# B&R Automation Studio project MotionTestBenchMaster (part 25)

#### Types.typ - Local data types
```iecst
TYPE
	MNM_AdjustmentStep :
		( (*V4.A.A.1.7.0*)
		MNM_AdjWaitStart := 100,
		MNM_AdjHornBlow := 110,
		MNM_AdjAxisStopping := 140,
		MNM_AdjFillerFootbarSettingPos := 200,
		MNM_AdjRinserFootbarSettingPos := 210,
		MNM_AdjDoserFootbarSettingPos := 220,
		MNM_AdjCapperSettingPos := 230,
		MNM_AdjCrownerSettingPos := 240,
		MNM_AdjCapGreasingSettingPos := 250, (*V4.A.A.1.7.0*)
		MNM_AdjAxisStart := 300,
		MNM_AdjAxisWaitStop := 310,
		MNM_AdjAxisPosStart := 400,
		MNM_AdjAxisPosWaitStop := 410,
		MNM_AdjAxisStopped := 500,
		MNM_AdjFault := 9999
		);
	MNM_AutoStep :
		(
		MNM_AutoWaitStart := 100,
		MNM_AutoHornBlow := 110,
		MNM_AutoMachineStart := 120,
		MNM_AutoMachineRunningEmpty := 131,
		MNM_AutoMachineRunningFull := 132,
		MNM_AutoMachineRunning := 133,
		MNM_AutoMachineColceaPashing := 134,
		MNM_AutoMachineStarWheel2Phasing := 137,
		MNM_AutoMachineRinserPashing := 136,
		MNM_AutoMachineStarWheel1Pashing := 135,
		MNM_AutoMachineStopping := 140,
		MNM_AutoSmr1OpHornBlow := 210,
		MNM_AutoSmr1OpMachineStart := 220,
		MNM_AutoSmr1OpMachineStopping := 240,
		MNM_AutoVortexCalibIdle := 300,
		MNM_AutoVortexCalibHornBlow := 310,
		MNM_AutoVortexCalibPosStart := 320,
		MNM_AutoVortexCalibPosWaitStop := 340,
		MNM_AutoStepFmcHornBlow := 410,
		MNM_AutoStepFmcStart := 420,
		MNM_AutoStepFmcWaitStop := 440,
		MNM_AutoStepHornBlow := 510,
		MNM_AutoStepStart := 520,
		MNM_AutoStepWaitStop := 540,
		MNM_AutoFootboardHornBlow := 610,
		MNM_AutoFootboardStart := 620,
		MNM_AutoFootboardWaitStop := 640,
		MNM_AutoCapperPosHornBlow := 710,
		MNM_AutoCapperPosStart := 720,
		MNM_AutoCapperPosWaitStop := 740,
		MNM_AutoCapperPosWaitStopAux := 741, (*V4.A.A.1.6.12h*)
		MNM_AutoCapperFinePosStart := 750,
		MNM_AutoCapperFinePosWaitStop := 760,
		MNM_AutoFillingValvePosHornBlow := 810,
		MNM_AutoFillingValvePosStart := 820,
		MNM_AutoFillingValvePosWaitStop := 830,
		MNM_AutoCheckFillerInletHorn := 1010,
		MNM_AutoCheckFillerInletStart := 1011,
		MNM_AutoCheckFillerInletStop := 1012,
		MNM_AutoCheckFillerTangencyHorn := 1020,
		MNM_AutoCheckFillerTangencyStart := 1021,
		MNM_AutoCheckFillerTangencyStop := 1022,
		MNM_AutoCheckFillerOutletHorn := 1030,
		MNM_AutoCheckFillerOutletStart := 1031,
		MNM_AutoCheckFillerOutletStop := 1032,
		MNM_AutoCheckCapsReleaseHorn := 1040,
		MNM_AutoCheckCapsReleaseStart := 1041,
		MNM_AutoCheckCapsReleaseStop := 1042,
		MNM_AutoFillerHalfPosConfig := 1043, (*v999*)
		MNM_AutoFillerHalfPosHornBlow := 1044, (*v999*)
		MNM_AutoFillerHalfAxisStart := 1045, (*v999*)
		MNM_AutoFillerHalfWaitStop := 1046, (*v999*)
		MNM_AutoFillerHalfStopped := 1047, (*v999*)
		MNM_AutoFillerReversePosConfig := 1048, (*v999*)
		MNM_AutoFillerReversePosHornBlow := 1049, (*v999*)
		MNM_AutoFillerReverseAxisStart := 1050, (*v999*)
		MNM_AutoFillerReverseWaitStop := 1051, (*v999*)
		MNM_AutoFillerReverseStopped := 1052, (*v999*)
		MNM_AutoFillSecondHalfPosConfig := 1053,
		MNM_AutoFillSecondHalfRevPosConf,
		MNM_AutoFault := 9999
		);
	MNM_AutoCombiStep :
		(
		MNM_AutoCombiInit := 0,
		MNM_AutoCombiBFWaitStart := 100,
		MNM_AutoCombiBLFWaitStart := 101,
		MNM_AutoCombiBAFWaitStart := 102, (*V4.A.A.1.7.0*)
		MNM_AutoCombiHornBlow := 110,
		MNM_AutoCombiSyncroStart := 120,
		MNM_AutoCombiMachineReadyToRun := 121,
		MNM_AutoCombiMachineRunningFull := 131,
		MNM_AutoCombiMachineRunningEmpty := 132,
		MNM_AutoCombiMachineFixEmptying := 135,
		MNM_AutoCombiMachineStopping := 140,
		MNM_AutoCombiFault := 9999
		);
	MNM_JogStep :
		(
		MNM_JogWaitStart := 400,
		MNM_JogHornBlow := 410,
		MNM_JogMachineStart := 420,
		MNM_JogMachineRunning := 430,
		MNM_JogMachineStopping := 440,
		MNM_JogFault := 9999
		);
	MNM_JogCombiStep :
		(
		MNM_JogCombiWaitStart := 400,
		MNM_JogCombiHornBlow := 410,
		MNM_JogCombiSyncroStart := 420,
		MNM_JogCombiMachineReadyToRun := 421,
		MNM_JogCombiMachineStart := 422,
		MNM_JogCombiMachineRunning := 430,
		MNM_JogCombiMachineStopping := 440,
		MNM_JogCombiFault := 9999
		);
	MNM_MultiStep :
		(
		MNM_MultiModeSelection := 0,
		MNM_MultiAutoWaitStart := 100,
		MNM_MultiAutoHornBlow := 110,
		MNM_MultiAutoMachineStart := 120,
		MNM_MultiAutoMachineRunning := 130,
		MNM_MultiAutoMachineStopping := 140,
		MNM_MultiVortexCalibIdle := 300,
		MNM_MultiVortexCalibHornBlow := 310,
		MNM_MultiVortexCalibPosStart := 320,
		MNM_MultiVortexCalibPosWaitStop := 340,
		MNM_MultiStepFmcHornBlow := 410,
		MNM_MultiStepFmcStart := 420,
		MNM_MultiStepFmcWaitStop := 440,
		MNM_MultiStepHornBlow := 510,
		MNM_MultiStepStart := 520,
		MNM_MultiStepWaitStop := 540,
		MNM_MultiFootboardHornBlow := 610,
		MNM_MultiFootboardStart := 620,
		MNM_MultiFootboardWaitStop := 640,
		MNM_MultiCapperPosHornBlow := 710,
		MNM_MultiCapperPosStart := 720,
		MNM_MultiCapperPosWaitStop := 740,
		MNM_MultiCapperFinePosStart := 750,
		MNM_MultiCapperFinePosWaitStop := 760,
		MNM_MultiJogWaitStart := 1400,
		MNM_MultiJogHornBlow := 1410,
		MNM_MultiJogMachineStart := 1420,
		MNM_MultiJogMachineRunning := 1430,
		MNM_MultiJogMachineStopping := 1440,
		MNM_MultiSlowMotionWaitStart := 1500,
		MNM_MultiSlowMotionHornBlow := 1510,
		MNM_MultiSlowMotionStart := 1520,
		MNM_MultiSlowMotionRunning := 1530,
		MNM_MultiSlowMotionStopping := 1540,
		MNM_MultiFault := 9999
		);
	MNM_InletConveyorVFD :
		( (*1.6(*Master nuovo*)
		MNM_InCvrIdle := 0,
		MNM_InCvrAuto := 100,
		MNM_InCvrAutoOption := 110,
		MNM_InCvrAutoFixSpeed := 210,
		MNM_InCvrAutoRampDown := 300,
		MNM_InCvrCleaning := 400,
		MNM_InCvrFault := 9999
		);
	MNM_OutletConveyorVFD :
		( (*1.6*)
		MNM_OutCvrIdle := 0,
		MNM_OutCvrAuto := 100,
		MNM_OutCvrAutoOption := 110,
		MNM_OutCvrAutoFixSpeed := 210,
		MNM_OutCvrAutoRampDown := 300,
		MNM_OutCvrCleaning := 400,
		MNM_OutCvrFault := 9999
		);
	VAR_FixSpeed_Type : 	STRUCT
		Module : USINT; (*0: All Module (Only coupled)
1: Inlet module
2: Filler module
3: Outlet module
9: All module (Uncupled) (Not interruptible)*)
		Interruptible : BOOL;
		Req : BOOL;
		Value : REAL;
		Reached : BOOL;
		CmpMode : USINT;
		Active : BOOL;
	END_STRUCT;
	VAR_ModuleSpeed_Type : 	STRUCT
		Machine : REAL;
		Inlet : REAL;
		Filler : REAL;
		Outlet : REAL;
	END_STRUCT;
END_TYPE
```

#### MNM_Devices.var - Local variables
```iecst
(*MOTORS*)
VAR
	_InCvrFC280 : Motor_FC280_Vfd;(*Master nuovo*)
	_OutCvrFC280 : Motor_FC280_Vfd; (*Outfeed Conveyor*)
	_InCvr : Motor_Vfd;(*Master nuovo*)
	_OutCvr : Motor_Vfd; (*Outfeed Conveyor*)
END_VAR
(*DIGITAL INSTRUMENTS*)
VAR
	_241DSE : Digital_Obj; (*Spot safety*)
	_230DSE : Digital_Obj; (*Spot safety*)
	_236DSE : Digital_Obj; (*Outlet obstructed*)
END_VAR
(*INLET CANS SENSOR*)
VAR
	InletSafetyLow1 : Digital_Obj;
	InletSafetyHigh1 : Digital_Obj;
	InletSafetyLow2 : Digital_Obj;
	InletSafetyHigh2 : Digital_Obj;
END_VAR
(*MOTORS FANS*)
(*Filler*)
VAR
	FillerFanMain : MotionFan_Obj;
	FillerFanIn1 : MotionFan_Obj;
	FillerFanIn2 : MotionFan_Obj;
	FillerFanIn3 : MotionFan_Obj;
	FillerFanIn4 : MotionFan_Obj;
	FillerFanIn5 : MotionFan_Obj;
	FillerFanIn6 : MotionFan_Obj;
	FillerFanIn7 : MotionFan_Obj;
	FillerFanIn8 : MotionFan_Obj;
	FillerFanIn9 : MotionFan_Obj;
	FillerFanIn10 : MotionFan_Obj;
	FillerFanOut1 : MotionFan_Obj;
	FillerFanOut2 : MotionFan_Obj;
	FillerFanOut3 : MotionFan_Obj;
	FillerFanOut4 : MotionFan_Obj;
	FillerFanOut5 : MotionFan_Obj;
END_VAR
(*Seamer*)
VAR
	OutletFanMain : MotionFan_Obj;
	OutletFanIn1 : MotionFan_Obj;
	OutletFanIn2 : MotionFan_Obj;
	OutletFanIn3 : MotionFan_Obj;
	OutletFanIn4 : MotionFan_Obj;
	OutletFanOut1 : MotionFan_Obj;
	OutletFanOut2 : MotionFan_Obj;
	OutletFanOut3 : MotionFan_Obj;
	OutletFanOut4 : MotionFan_Obj;
END_VAR
```

#### Package Logical/05_MNM/MNM/0520_InletConveyor - Conveyor: motori nastri Ingresso Macchina

#### InletConveyorVar_VFD.st
```iecst
ACTION InletConveyorVar_VFD:
//	VAR_MNM_ConveyorProduction	:= MC_InputOutput.Network.Filler.Status.ModuleRunning OR OPS.DataOut.FlrModeSelectorJog;
//	VAR_MNM_ConveyorClean		:= COP.DataOut.RcpActive;
END_ACTION
```

#### InletConveyorSeq_VFD.st
```iecst
ACTION InletConveyorSeq_Run_VFD:

	VAR_MNM_InCvrAlarm			:= ALR[7029].Active OR ALR[7031].Active OR ALR[7032].Active;
	_InCvrFC280.IN_AutoCnd			:= FALSE;
	_InCvrFC280.IN_AutoSpeed		:= 0.0;

	//Speed Linearization
	FB_ScalConveyorInlet(
	x	:= MC_InputOutput.Network.Machine.Status.ActualSpeed,
	x1	:= 0.0,
	y1	:= 0.0,
	x2	:= MC_InputOutput.Network.Machine.Status.MachineMaxSpeed * 1.1,
	y2	:= _InCvrFC280.IN_FrequencyMax + (_InCvrFC280.IN_FrequencyMax * HMI_PAR_1._160 / 100.0) * 1.1,
	);

	//State Management
	CASE VAR_MNM_InletConveyorSeq_VFD OF
		MNM_InCvrIdle:
			IF MNM.DataOut.MachineRunning AND NOT COP.DataOut.RcpActive AND NOT OPS.DataOut.FlrModeSelectorAdjustment THEN
				VAR_MNM_InletConveyorSeq_VFD := MNM_InCvrAuto;
			ELSIF COP.DataOut.RcpActive THEN
				_InCvrFC280.IN_AutoCnd	:= TRUE;
				VAR_MNM_InletConveyorSeq_VFD := MNM_InCvrCleaning;
			ELSIF VAR_MNM_InCvrAlarm THEN
				VAR_MNM_InletConveyorSeq_VFD := MNM_InCvrFault;
			END_IF

		MNM_InCvrAuto:

			_InCvrFC280.IN_AutoCnd		:= FB_ScalConveyorInlet.y>0.0;
			_InCvrFC280.IN_AutoSpeed	:= FB_ScalConveyorInlet.y;

			IF NOT MNM.DataOut.MachineRunning THEN
				VAR_MNM_InletConveyorSeq_VFD	:= MNM_InCvrIdle;
			ELSIF VAR_MNM_InCvrAlarm THEN
				VAR_MNM_InletConveyorSeq_VFD	:= MNM_InCvrFault;
			END_IF

		MNM_InCvrCleaning:
			_InCvrFC280.IN_AutoCnd		:= MC_InputOutput.Network.Machine.Status.MachineRunning;
			_InCvrFC280.IN_AutoSpeed	:= 10.0;

			IF NOT COP.DataOut.RcpActive THEN
				VAR_MNM_InletConveyorSeq_VFD	:= MNM_InCvrIdle;
			ELSIF VAR_MNM_InCvrAlarm THEN
				VAR_MNM_InletConveyorSeq_VFD	:= MNM_InCvrFault;
			END_IF

		MNM_InCvrFault:
			IF AID.DataOut.Reset THEN
				VAR_MNM_InletConveyorSeq_VFD := MNM_InCvrIdle;
			END_IF
	END_CASE

	TMR_TON_MNM_InCvrFix	(IN:= (VAR_MNM_InletConveyorSeq_VFD = MNM_InCvrAutoFixSpeed), PT := t#120s);
	TMR_TON_MNM_InCvrRamp	(IN:= (VAR_MNM_InletConveyorSeq_VFD = MNM_InCvrAutoRampDown), PT := t#5s);
END_ACTION
```

#### InletConveyorMotors_VFD.st
```iecst
ACTION InletConveyorMotors_VFD:
//	_InCvr(//Management with FC302
//	IN_Enable		:= OPS.DataOut.EnableDrive,
//	IN_AutoCnd		:= _InCvr.IN_AutoCnd,
//	IN_FrequencyMin	:= 0.0,
//	IN_FrequencyMax	:= 100.0,
//	IN_ManEn		:= TRUE,
//	IN_MaskEn		:= TRUE,
//	IN_Reset		:= AID.DataOut.Reset,
//	IN_HMIAutoForce	:= NOT HMI_SS2P[SS2P_HMI_DeviceEnable].ON,
//	IN_QuickStopCmd	:= NOT OPS.DataOut.EnableDrive,
//	IN_CoastingCmd	:= FALSE,
//	IN_ScaleMax		:= 100.0,
//	HMI_Danfoss		:= HMI_VFD_InCvr,
//	HMI_Motor		:= HMI_InCvr,
//	IO_Danfoss		:= IO_VFD_InCvr,
//	IO_Motor		:= IO_InCvr
//	);

	_InCvrFC280(
	IN_Enable		:= OPS.DataOut.EnableDrive,
	IN_AutoCnd		:= _InCvrFC280.IN_AutoCnd,
	IN_FrequencyMin	:= 0.0,
	IN_FrequencyMax	:= 100.0,
	IN_ManEn		:= TRUE,
	IN_MaskEn		:= TRUE,
	IN_Reset		:= AID.DataOut.Reset,
	IN_HMIAutoForce	:= NOT HMI_SS2P[SS2P_HMI_DeviceEnable].ON,
	IN_QuickStopCmd	:= NOT OPS.DataOut.EnableDrive,
	IN_CoastingCmd	:= FALSE,
	IN_ScaleMax		:= 100.0,
	HMI_Danfoss		:= HMI_VFD_InCvr,
	HMI_Motor		:= HMI_InCvr,
	IO_DanfossFC280	:= IO_VFD_InCvrFC280,
	IO_MotorFC280	:= IO_InCvrFC280
	);

END_ACTION
```

#### InletConveyorDataOut_VFD.st
```iecst
ACTION InletConveyorDataOut_VFD:
//	IF _InCvr.OUT_ActualFrequency > 0 THEN
//		MNM.DataOut.OutletSpeed := (((_InCvr.OUT_ActualFrequency / 100.0) * MC_InputOutput.Network.Machine.Status.ActualSpeed) / 60.0);
//	ELSE
//		MNM.DataOut. := 0.0 ;
//	END_IF
END_ACTION
```

#### InletConveyorAlarm_VFD.st
```iecst
ACTION InletConveyorAlarm_VFD:
//
//	ALR[7029].Active		:= _InCvr.OUT_OverloadFault;//Management with FC302
//	ALR[7031].Active		:= _InCvr.OUT_IsolatedFault;//Management with FC302
//	ALR[7032].Active		:= _InCvr.OUT_DriveFault;//Management with FC302

	ALR[7029].Active		:= _InCvrFC280.OUT_OverloadFault;
	ALR[7031].Active		:= _InCvrFC280.OUT_IsolatedFault;
	ALR[7032].Active		:= _InCvrFC280.OUT_DriveFault;
END_ACTION
```

#### InletConveyorHMI.st
```iecst
ACTION InletConveyorHMI:
	IF TNK.DataOut.ProdMode AND NOT TNK.DataOut.StartUp THEN
		HMI_ContainerFallInlet1	:= (InletSafetyLow1.OUT AND NOT InletSafetyHigh1.OUT) OR (NOT InletSafetyLow1.OUT AND InletSafetyHigh1.OUT);
		HMI_ContainerFallInlet2	:= (InletSafetyLow2.OUT AND NOT InletSafetyHigh2.OUT) OR (NOT InletSafetyLow2.OUT AND InletSafetyHigh2.OUT);
		HMI_NoContainerInlet1	:= (NOT InletSafetyLow1.OUT AND NOT InletSafetyHigh1.OUT);
		HMI_NoContainerInlet2	:= (NOT InletSafetyLow2.OUT AND NOT InletSafetyHigh2.OUT);
	ELSE
		HMI_ContainerFallInlet1	:= FALSE;
		HMI_ContainerFallInlet2	:= FALSE;
		HMI_NoContainerInlet1	:= FALSE;
		HMI_NoContainerInlet1	:= FALSE;
	END_IF
END_ACTION
```

#### InletConveyorAlarm.st
```iecst
ACTION InletConveyorAlarm:
	IF InletSafetyLow1.OUT_OffDelayed AND InletSafetyHigh1.OUT_OffDelayed AND TNK.DataOut.ProdMode AND NOT TNK.DataOut.StartUp AND CvoFlr.InfeedConveyorRunning THEN
		ALR[4618].Active	:= TRUE;   //TRUE; //COLLAUDO
	ELSE
		ALR[4618].Active	:= FALSE;
	END_IF

	IF InletSafetyLow2.OUT_OffDelayed AND InletSafetyHigh2.OUT_OffDelayed AND TNK.DataOut.ProdMode AND NOT TNK.DataOut.StartUp THEN
		ALR[4619].Active	:= TRUE;
	ELSIF AID.DataOut.Reset THEN
		ALR[4619].Active	:= FALSE;
	END_IF

	IF SFT.DataOut.ContainersBlock1 THEN
		IF TON_ContainerInletSafety1.Q AND TNK.DataOut.ProdMode AND NOT TNK.DataOut.StartUp THEN
			ALR[4620].Active	:= TRUE;
		ELSIF AID.DataOut.Reset THEN
			ALR[4620].Active	:= FALSE;
		END_IF
	ELSE
		IF ((InletSafetyLow1.OUT AND NOT InletSafetyHigh1.OUT) OR (NOT InletSafetyLow1.OUT AND InletSafetyHigh1.OUT)) AND TNK.DataOut.ProdMode AND NOT TNK.DataOut.StartUp THEN
			ALR[4620].Active	:= TRUE;
		ELSIF IO_PB_ResetInlet1.ON THEN
			ALR[4620].Active	:= FALSE;
		END_IF
	END_IF
	TON_ContainerInletSafety1.IN := ((InletSafetyLow1.OUT AND NOT InletSafetyHigh1.OUT) OR (NOT InletSafetyLow1.OUT AND InletSafetyHigh1.OUT));
	TON_ContainerInletSafety1.PT := REAL_TO_TIME((1/(MC_InputOutput.Network.Machine.Status.ActualSpeed/3600))*1000 );
	TON_ContainerInletSafety1();

	IO_PB_ResetInlet1.LampON := ALR[4620].Active AND AID.DataOut.Blink1Hz;

	IF ((InletSafetyLow2.OUT AND NOT InletSafetyHigh2.OUT) OR (NOT InletSafetyLow2.OUT AND InletSafetyHigh2.OUT)) AND TNK.DataOut.ProdMode AND NOT TNK.DataOut.StartUp THEN
		ALR[4621].Active	:= TRUE;
	ELSIF IO_PB_ResetInlet2.ON THEN
		ALR[4621].Active	:= FALSE;
	END_IF

	MNM.DataOut.LackInlet1 := ALR[4618].Active OR ALR[4620].Active;
	MNM.DataOut.LackInlet2 := ALR[4619].Active OR ALR[4621].Active;

	ALR[4600].Active	:= NOT IO_LimitTorqueBlowerTransfer.DI_Input;

END_ACTION
```

#### InletConveyor_Hardware_CFG.st
```iecst
ACTION InletConveyor_Hardware_CFG:
	(*****SENSORS*****)
	InletSafetyLow1.IN_ConfigPresent	:= TRUE;
	InletSafetyLow1.IN_OffDelay			:= t#200ms;
	InletSafetyLow1.IN_OnDelay			:= t#200ms;
	InletSafetyLow1.IN_SwitchDelay		:= t#0ms;

	InletSafetyHigh1.IN_ConfigPresent	:= TRUE;
	InletSafetyHigh1.IN_OffDelay		:= t#200ms;
	InletSafetyHigh1.IN_OnDelay			:= t#200ms;
	InletSafetyHigh1.IN_SwitchDelay		:= t#0ms;

	InletSafetyLow2.IN_ConfigPresent	:= FALSE;
	InletSafetyLow2.IN_OffDelay			:= t#200ms;
	InletSafetyLow2.IN_OnDelay			:= t#200ms;
	InletSafetyLow2.IN_SwitchDelay		:= t#0ms;

	InletSafetyHigh2.IN_ConfigPresent	:= FALSE;
	InletSafetyHigh2.IN_OffDelay		:= t#200ms;
	InletSafetyHigh2.IN_OnDelay			:= t#200ms;
	InletSafetyHigh2.IN_SwitchDelay		:= t#0ms;

//	(*****MOTORS*****)//For Inverter Model FC302, old Hardware standard
//	_InCvr.IN_ConfigPresent			:= FALSE;
//	_InCvr.IN_SafetyCtrlEn			:= TRUE;
//	_InCvr.IN_Simulation			:= FALSE;
//	_InCvr.IN_FBKDelay				:= t#1200ms;

	(*****MOTORS*****)//For Inverter Model FC280, new Hardware standard
	_InCvrFC280.IN_ConfigPresent	:= TRUE;
	_InCvrFC280.IN_SafetyCtrlEn		:= TRUE;
	_InCvrFC280.IN_Simulation		:= FALSE;
	_InCvrFC280.IN_FBKDelay			:= t#1200ms;

END_ACTION
```

#### InletConveyorDigitalIn.st
```iecst
ACTION InletConveyorDigitalIn:
	InletSafetyLow1(
	IN_ConfigPresent	:= InletSafetyLow1.IN_ConfigPresent,
	IN_Alarm			:= TRUE,
	IN_Reset			:= AID.DataOut.Reset,
	IO					:= IO_InletSafetyLow1,
	HMI					:= HMI_InletSafetyLow1
	);

	InletSafetyHigh1(
	IN_ConfigPresent	:= InletSafetyHigh1.IN_ConfigPresent,
	IN_Alarm			:= TRUE,
	IN_Reset			:= AID.DataOut.Reset,
	IO					:= IO_InletSafetyHigh1,
	HMI					:= HMI_InletSafetyHigh1
	);

	InletSafetyLow2(
	IN_ConfigPresent	:= InletSafetyLow2.IN_ConfigPresent,
	IN_Alarm			:= TRUE,
	IN_Reset			:= AID.DataOut.Reset,
	IO					:= IO_InletSafetyLow2,
	HMI					:= HMI_InletSafetyLow2
	);

	InletSafetyHigh2(
	IN_ConfigPresent	:= InletSafetyHigh2.IN_ConfigPresent,
	IN_Alarm			:= TRUE,
	IN_Reset			:= AID.DataOut.Reset,
	IO					:= IO_InletSafetyHigh2,
	HMI					:= HMI_InletSafetyHigh2
	);
END_ACTION
```

#### InletConveyorInterchange.st - not listed in the package file held
```iecst
ACTION InletConveyorInterchange:

END_ACTION
```

#### Package Logical/05_MNM/MNM/0530_OutletConveyor - Conveyor: motori nastri Uscita Macchina

#### OutletConveyor_Hardware_CFG.st
```iecst
ACTION OutletConveyor_Hardware_CFG:
	(*****MOTORS*****)//For Inverter Model FC302, old Hardware standard
//	_OutCvr.IN_ConfigPresent	:= FALSE;
//	_OutCvr.IN_SafetyCtrlEn		:= TRUE;
//	_OutCvr.IN_Simulation		:= FALSE;
//	_OutCvr.IN_FBKDelay			:= t#1200ms;

	(*****MOTORS*****)//For Inverter Model FC280, new Hardware standard
	_OutCvrFC280.IN_ConfigPresent	:= TRUE;
	_OutCvrFC280.IN_SafetyCtrlEn		:= TRUE;
	_OutCvrFC280.IN_Simulation		:= FALSE;
	_OutCvrFC280.IN_FBKDelay			:= t#1200ms;
	(*****SENSORS*****)
	// Exit Spot #1
	_230DSE.IN_ConfigPresent	:= TRUE;
	_230DSE.IN_Alarm			:= TRUE;
	_230DSE.IN_OffDelay			:= t#0s;
	_230DSE.IN_OnDelay			:= t#500ms;
	_230DSE.IN_SwitchDelay		:= t#0ms;
	// Outlet Conveyor Guide
	_236DSE.IN_ConfigPresent	:= FALSE;
	_236DSE.IN_Alarm			:= TRUE;
	_236DSE.IN_OffDelay			:= t#0s;
	_236DSE.IN_OnDelay			:= t#500ms;
	_236DSE.IN_SwitchDelay		:= t#0ms;

END_ACTION
```

#### OutletConveyorVar_VFD.st
```iecst
ACTION OutletConveyorVar_VFD:
	VAR_MNM_ConveyorProduction	:= MNM.DataOut.MachineRunning AND NOT COP.DataOut.RcpActive OR OPS.DataOut.FlrModeSelectorJog; //Montanarini: a Heuft serve il nastro in movimento quando la macchina gira	---	NOT SFT.DataOut.OutletConveyorEmpty OR NOT SFT.DataOut.MachineEmpty OR OPS.DataOut.FlrModeSelectorJog;
	VAR_MNM_ConveyorClean		:= COP.DataOut.RcpActive;
END_ACTION
```

#### OutletConveyorSeq_VFD.st
```iecst
ACTION OutletConveyorSeq_Run_VFD:
	//VAR_MNM_OutCvrAlarm			:= 	AID.DataOut.ALR.Bit.ALR_MS_NormalStop OR AID.DataOut.ALR.Bit.ALR_MS_QuickStop OR AID.DataOut.ALR.Bit.ALR_MS_NormalWithJog OR
	//								AID.DataOut.ALR.Bit.ALR_MS_QuickWithJog OR AID.DataOut.ALR.Bit.ALR_CSR_StopAfterEmptying;

	VAR_MNM_OutCvrAlarm		:= ALR[4633].Active OR ALR[4638].Active OR ALR[7039].Active OR ALR[7041].Active OR ALR[7042].Active;
	_OutCvr.IN_AutoCnd			:= FALSE;
	_OutCvr.IN_AutoSpeed		:= 0.0;

	//VAR_MNM_OptionNoGripper -> To be setted
	VAR_MNM_OptionNoGripper := TRUE;//VAR_MNM_OptionNoGripper := TRUE means that the outlet starwheel is without gripper //V4.A.A.1.6.6
									//VAR_MNM_OptionNoGripper := FALSE means that the outlet starwheel is with gripper //V4.A.A.1.6.6

	//Speed Linearization
	FB_ScalConveyor(
	x	:= MC_InputOutput.Network.Machine.Status.ActualSpeed,
	x1	:= 0.0,
	y1	:= 0.0,
	x2	:= MC_InputOutput.Network.Machine.Status.MachineMaxSpeed * 1.1,
	y2	:= _OutCvrFC280.IN_FrequencyMax + (_OutCvrFC280.IN_FrequencyMax * HMI_PAR_1._162 / 100.0) * 1.1,
	);

	//Speed Limit Threshold
	VAR_MNM_OutCvrFixSpeedLimit := MC_InputOutput.Network.Machine.Status.ActualSpeed > 10000.0;

	//Fixed Speed Calculation
	IF EDGEPOS(VAR_MNM_OutCvrFixSpeedLimit) OR EDGENEG(VAR_MNM_OutCvrFixSpeedLimit) THEN
		VAR_MNM_OutCvrFixSpeed		:= FB_ScalConveyor.y;
	END_IF

	//Fixed Speed Calculation in case of data loss
	IF VAR_MNM_OutCvrFixSpeed = 0 THEN
		VAR_MNM_OutCvrFixSpeed		:= 20.0;
	END_IF

	//State Management
	CASE VAR_MNM_OutletConveyorSeq_VFD OF
		MNM_OutCvrIdle:
			IF VAR_MNM_ConveyorProduction THEN//v1.61
				VAR_MNM_OutletConveyorSeq_VFD := MNM_OutCvrAuto;
			ELSIF VAR_MNM_ConveyorClean THEN
				_OutCvr.IN_AutoCnd	:= TRUE;
				VAR_MNM_OutletConveyorSeq_VFD := MNM_OutCvrCleaning;
			ELSIF VAR_MNM_OutCvrAlarm THEN
				VAR_MNM_OutletConveyorSeq_VFD := MNM_OutCvrFault;
			END_IF

		MNM_OutCvrAuto:

			_OutCvr.IN_AutoCnd		:= FB_ScalConveyor.y>0.0;//V4.A.A.1.6.6
			_OutCvr.IN_AutoSpeed	:= FB_ScalConveyor.y;

			IF NOT VAR_MNM_ConveyorProduction THEN
				VAR_MNM_OutletConveyorSeq_VFD	:= MNM_OutCvrIdle;
			ELSIF VAR_MNM_ConveyorProduction AND VAR_MNM_OptionNoGripper AND VAR_MNM_OutCvrFixSpeedLimit THEN//v1.61
				VAR_MNM_OutletConveyorSeq_VFD := MNM_OutCvrAutoOption;//v1.61
			ELSIF VAR_MNM_OutCvrAlarm THEN
				VAR_MNM_OutletConveyorSeq_VFD	:= MNM_OutCvrFault;
			END_IF

		MNM_OutCvrAutoOption:

			_OutCvr.IN_AutoCnd		:= FB_ScalConveyor.y>0.0;//V4.A.A.1.6.6
			_OutCvr.IN_AutoSpeed	:= FB_ScalConveyor.y;

			IF NOT VAR_MNM_ConveyorProduction OR (NOT VAR_MNM_OutCvrFixSpeedLimit AND NOT MC_InputOutput.Network.Machine.Commands.MachineStart) THEN
				VAR_MNM_OutletConveyorSeq_VFD	:= MNM_OutCvrAutoFixSpeed;
			ELSIF VAR_MNM_OutCvrAlarm THEN
				VAR_MNM_OutletConveyorSeq_VFD	:= MNM_OutCvrFault;
			END_IF

		MNM_OutCvrAutoFixSpeed:
			_OutCvr.IN_AutoCnd			:= FB_ScalConveyor.y>0.0;//V4.A.A.1.6.6
			TMR_TON_MNM_OutCvrFix.IN 	:= TRUE;

			IF MC_InputOutput.Network.Machine.Commands.MachineStart OR VAR_MNM_OutCvrFixSpeedLimit THEN
				_OutCvr.IN_AutoSpeed 		:= FB_ScalConveyor.y;
			ELSIF NOT VAR_MNM_OutCvrFixSpeedLimit AND NOT MC_InputOutput.Network.Machine.Commands.MachineStart THEN
				_OutCvr.IN_AutoSpeed 		:= VAR_MNM_OutCvrFixSpeed;
			END_IF

			IF MC_InputOutput.Network.Machine.Commands.MachineStart AND VAR_MNM_ConveyorProduction THEN
				VAR_MNM_OutletConveyorSeq_VFD	:= MNM_OutCvrAuto;
			ELSIF TMR_TON_MNM_OutCvrFix.Q THEN
				VAR_MNM_OutletConveyorSeq_VFD	:= MNM_OutCvrAutoRampDown;
				VAR_MNM_OutCvrRampDwStart		:= _OutCvr.IN_AutoSpeed;
			ELSIF VAR_MNM_OutCvrAlarm THEN
				VAR_MNM_OutletConveyorSeq_VFD	:= MNM_OutCvrFault;
			END_IF

		MNM_OutCvrAutoRampDown:
			_OutCvr.IN_AutoCnd			:= TRUE;
			_OutCvr.IN_AutoSpeed 		:= VAR_MNM_OutCvrRampDwStart -
											(VAR_MNM_OutCvrRampDwStart * (UDINT_TO_REAL(TIME_TO_UDINT(TMR_TON_MNM_OutCvrRamp.ET))) /
											(UDINT_TO_REAL(TIME_TO_UDINT(TMR_TON_MNM_OutCvrRamp.PT))));
			TMR_TON_MNM_OutCvrRamp.IN 	:= TRUE;

			IF MC_InputOutput.Network.Machine.Commands.MachineStart AND VAR_MNM_ConveyorProduction THEN
				VAR_MNM_OutletConveyorSeq_VFD	:= MNM_OutCvrAuto;
			ELSIF TMR_TON_MNM_OutCvrRamp.Q THEN
				VAR_MNM_OutletConveyorSeq_VFD	:= MNM_OutCvrIdle;
			ELSIF VAR_MNM_OutCvrAlarm THEN
				VAR_MNM_OutletConveyorSeq_VFD	:= MNM_OutCvrFault;
			END_IF

		MNM_OutCvrCleaning:
			_OutCvr.IN_AutoCnd		:= MC_InputOutput.Network.Machine.Status.MachineRunning;
			_OutCvr.IN_AutoSpeed	:= 10.0;

			IF NOT VAR_MNM_ConveyorClean THEN
				VAR_MNM_OutletConveyorSeq_VFD	:= MNM_OutCvrIdle;
			ELSIF VAR_MNM_OutCvrAlarm THEN
				VAR_MNM_OutletConveyorSeq_VFD	:= MNM_OutCvrFault;
			END_IF

		MNM_OutCvrFault:
			IF AID.DataOut.Reset THEN
				VAR_MNM_OutletConveyorSeq_VFD := MNM_OutCvrIdle;
			END_IF
	END_CASE

	TMR_TON_MNM_OutCvrFix	(IN:= (VAR_MNM_OutletConveyorSeq_VFD = MNM_OutCvrAutoFixSpeed), PT := t#120s);//<<Change this time to decide how long the conveyour runs after the last bottle or machine stop.
	TMR_TON_MNM_OutCvrRamp	(IN:= (VAR_MNM_OutletConveyorSeq_VFD = MNM_OutCvrAutoRampDown), PT := t#5s);
END_ACTION
```

#### OutletConveyorMotors_VFD.st
```iecst
ACTION OutletConveyorMotors_VFD:
//	_OutCvr(//Management with FC302
//	IN_Enable		:= OPS.DataOut.EnableDrive,
//	IN_AutoCnd		:= _OutCvr.IN_AutoCnd,
//	IN_FrequencyMin	:= 0.0,
//	IN_FrequencyMax	:= 100.0,
//	IN_ManEn		:= TRUE,
//	IN_MaskEn		:= TRUE,
//	IN_Reset		:= AID.DataOut.Reset,
//	IN_HMIAutoForce	:= NOT HMI_SS2P[SS2P_HMI_DeviceEnable].ON,
//	IN_QuickStopCmd	:= NOT OPS.DataOut.EnableDrive,
//	IN_CoastingCmd	:= FALSE,
//	IN_ScaleMax		:= 100.0,
//	HMI_Danfoss		:= HMI_VFD_OutCvr,
//	HMI_Motor		:= HMI_OutCvr,
//	IO_Danfoss		:= IO_VFD_OutCvr,
//	IO_Motor		:= IO_OutCvr
//	);

	_OutCvrFC280.IN_AutoCnd 	:= _OutCvr.IN_AutoCnd;
	_OutCvrFC280.IN_AutoSpeed	:= _OutCvr.IN_AutoSpeed;	//Montanarini: appoggio velocità

	_OutCvrFC280(
	IN_Enable		:= OPS.DataOut.EnableDrive,
	IN_AutoCnd		:= _OutCvrFC280.IN_AutoCnd,
	IN_FrequencyMin	:= 0.0,
	IN_FrequencyMax	:= 100.0,
	IN_ManEn		:= TRUE,
	IN_MaskEn		:= TRUE,
	IN_Reset		:= AID.DataOut.Reset,
	IN_HMIAutoForce	:= NOT HMI_SS2P[SS2P_HMI_DeviceEnable].ON,
	IN_QuickStopCmd	:= NOT OPS.DataOut.EnableDrive,
	IN_CoastingCmd	:= FALSE,
	IN_ScaleMax		:= 100.0,
	HMI_Danfoss		:= HMI_VFD_OutCvr,
	HMI_Motor		:= HMI_OutCvr,
	IO_DanfossFC280		:= IO_VFD_OutCvrFC280,
	IO_MotorFC280		:= IO_OutCvrFC280
	);

END_ACTION
```

#### OutletConveyorDataOut_VFD.st
```iecst
ACTION OutletConveyorDataOut_VFD:
	IF _OutCvrFC280.OUT_ActualFrequency > 0 THEN
		MNM.DataOut.OutletSpeed := (((_OutCvrFC280.OUT_ActualFrequency / 100.0) * MC_InputOutput.Network.Machine.Status.ActualSpeed) / 60.0);
	ELSE
		MNM.DataOut.OutletSpeed := 0.0 ;
	END_IF
END_ACTION
```

#### OutletConveyorAlarm_VFD.st
```iecst
ACTION OutletConveyorAlarm_VFD:
//	ALR[7039].Active		:= _OutCvr.OUT_OverloadFault;//Management with FC302
//	ALR[7041].Active		:= _OutCvr.OUT_IsolatedFault//Management with FC302
//	ALR[7042].Active		:= _OutCvr.OUT_DriveFault//Management with FC302

	ALR[7039].Active		:= _OutCvrFC280.OUT_OverloadFault;
	ALR[7041].Active		:= _OutCvrFC280.OUT_IsolatedFault;
	ALR[7042].Active		:= _OutCvrFC280.OUT_DriveFault;

	ALR[4638].Active	:= _236DSE.OUT_Alarm;
	ALR[4633].Active	:= _230DSE.OUT_Alarm;

END_ACTION
```

#### OutletConveyorMotors_Motion.st
```iecst
ACTION OutletConveyorMotors_Motion:
	MC_InputOutput.Network.Filler.Parameters.InletConveyorKs	:= HMI_PAR_1._160;
	MC_InputOutput.Network.Filler.Parameters.OutletConveyorKs	:= HMI_PAR_1._162;
	MC_InputOutput.Network.Outlet.Parameters.ConveyorKs		:= HMI_PAR_1._162;
END_ACTION
```

#### OutletConveyorAlarm_Motion.st
```iecst
ACTION OutletConveyorAlarm_Motion:
	IF NOT IO_OutCvr.DI_ManSwitchON THEN
		ALR[7041].Active	:= TRUE;
	ELSIF AID.DataOut.Reset THEN
		ALR[7041].Active	:= FALSE;
	END_IF

	ALR[4638].Active	:= _236DSE.OUT_Alarm;//v1.7.2
	ALR[4633].Active	:= _230DSE.OUT_Alarm;//v1.7.2

END_ACTION
```

#### OutletConveyorDataOut_Motion.st
```iecst
ACTION OutletConveyorDataOut_Motion:
	MNM.DataOut.OutletSpeed := ((MC_InputOutput.Network.Machine.Status.ActualSpeed / 60.0) * (1 + MC_InputOutput.Network.Outlet.Parameters.ConveyorKs / 100.0)) * LREAL_TO_REAL(CFG_MC.Mechanical.MachineStep / 1000.0) * 10.0;
END_ACTION
```

#### OutletConveyorDigitalIn.st
```iecst
ACTION OutletConveyorDigitalIn:
	_230DSE(
	IN_ConfigPresent	:= _230DSE.IN_ConfigPresent,
	IN_Reset			:= AID.DataOut.Reset,
	IN_MaskEn			:= FALSE,
	IN_WaitOn			:= TRUE,
	IN_AlarmOffReq		:= TRUE,
	IO					:= IO_230DSE,
	HMI					:= HMI_230DSE
	);

	_236DSE(
	IN_ConfigPresent	:= _236DSE.IN_ConfigPresent,
	IN_Reset			:= AID.DataOut.Reset,
	IN_MaskEn			:= FALSE,
	IN_WaitOn			:= TRUE,
	IN_AlarmOffReq		:= TRUE,
	IO					:= IO_236DSE,
	HMI					:= HMI_236DSE
	);
END_ACTION
```

#### OutletConveyorInterchange.st
```iecst
ACTION OutletConveyorInterchange:
(***************************      Alarms Standard        ****************************************)
	ALR[4626].Active	:= ((NOT CvoFlr.InfeedContainersLoadEnabled AND NOT CvoFlr.Req_Empty AND NOT SkdFlr.EndProduction) AND TNK.DataOut.ProdMode AND NOT TNK.DataOut.StartUp); //OR CvoFlr.Req_Empty;
	ALR[4629].Active	:= NOT CvoFlr.InfeedConveyorRunning AND TNK.DataOut.ProdMode AND NOT TNK.DataOut.StartUp;
	ALR[4632].Active	:= NOT CvoFlr.OutletConveyorRunning AND TNK.DataOut.ProdMode AND NOT TNK.DataOut.StartUp;
	ALR[4635].Active	:= CvoFlr.RejectTableFull AND TNK.DataOut.ProdMode AND NOT TNK.DataOut.StartUp;
	ALR[4636].Active	:= FALSE;//MasterBottle
	//ALR[4636].Active	:= CvoFlr.OutletConveyorLowSpeed AND TNK.DataOut.ProdMode AND NOT TNK.DataOut.StartUp;//PET(*Master nuovo*)
	ALR[4637].Active	:= NOT CvoFlr.OutletContainersLoadEnabled AND TNK.DataOut.ProdMode AND NOT TNK.DataOut.StartUp;
END_ACTION
```

#### OutletConveyorHMI.st
```iecst
ACTION OutletConveyorHMI:
	IF TNK.DataOut.ProdMode AND NOT TNK.DataOut.StartUp THEN
		HMI_OutletFull	:= CvoFlr.OutletConveyorLowSpeed OR NOT CvoFlr.OutletContainersLoadEnabled;
	ELSE
		HMI_OutletFull	:= FALSE;
	END_IF
END_ACTION
```

#### MNM_DataOut.st
```iecst
ACTION MNM_DataOut:
	MNM.DataOut.HornFlrRequest		:= VAR_MNM_HornFlrRequest;

	MNM.DataOut.ReadyForVortexCalib	:= VAR_MNM_AutoVortexCalibActive;

	MNM.DataOut.ReadyForCoupling	:= MC_InputOutput.Network.Machine.Status.EnableCombi;

	MNM.DataOut.FixSpeedRequest 	:= VAR_MNM_FixSpeedReq;

	MNM.DataOut.COPInletContBlockSpeedReached	:= VAR_FixSpeed[10].Reached;

	MNM.DataOut.MachineRunning		:= SEL(MC_InputOutput.Network.Machine.Status.MultiModalityActive, MC_InputOutput.Network.Machine.Status.MachineRunning, MC_InputOutput.Network.Filler.Status.ModuleRunning); //V1.0
	MNM.DataOut.RinserAxisDisabled    	:= MC_InputOutput.Network.Filler.Status.RinserAxisDisabled;//V4.A.A.1.7.0
	MNM.DataOut.DoserAxisDisabled		:= MC_InputOutput.Network.Filler.Status.DoserAxisDisabled;//v999hema
	MNM.DataOut.FillerAxisDisabled		:= MC_InputOutput.Network.Filler.Status.FillerAxisDisabled;//v999hema
	IF EDGEPOS(IO_PB_FlStart.ON)	OR EDGENEG(IO_PB_FlStop.ON)	THEN
		MNM.DataOut.OperatorPresence	:= 	TRUE;
	END_IF

END_ACTION
```

#### MNM_Alarm.st
```iecst
ACTION MNM_Alarm:

	ALR[7018].Active		:= (MC_InputOutput.Network.Machine.Status.ActualSpeed >
								(MC_InputOutput.Network.Machine.Status.MachineMaxSpeed + (MC_InputOutput.Network.Machine.Status.MachineMaxSpeed * 8.0 / 100.0))) AND MC_InputOutput.Network.Machine.Status.AutoCombiModalityActive;

	ALR[7019].Active		:= MC_InputOutput.Network.Machine.Status.ActualSpeed > (HMI_PAR_1._020 + (HMI_PAR_1._020 * 5.0 / 100.0));

	//v4 200.2.0 eliminata logica

	ALR[7155].Active	:= MC_InputOutput.Network.Machine.Exceptions.PowerSupplyLowMachineException; //V4.A.A.1.6.13
	ALR[7156].Active    := NOT IO_MNM_PowerSupply1Overload.DI_Input; //V4.A.A.1.6.13
	ALR[7157].Active	:= NOT IO_MNM_PowerSupply2Overload.DI_Input; //V4.A.A.1.6.13

	//V4.A.A.1.6.13
	ALR[7170].Active	:= (HMI_PAM_1._403 = 0) AND (HMI_201CPC.ConfigPresent OR HMI_202CPC.ConfigPresent);
	ALR[7171].Active	:= (HMI_PAM_1._407 = 0) AND CFG_Par.ClosingUnit.Capper.Present;
	ALR[7173].Active	:= (HMI_PAM_1._415 = 0) AND (HMI_PAO_2._176 <> 0);
	ALR[7174].Active 	:= (HMI_PAM_1._419 = 0) AND HMI_201CPB.ConfigPresent;
	ALR[7175].Active	:= (HMI_PAM_1._423 = 0) AND CFG_Par.ClosingUnit.Crowner.Present;
	ALR[7176].Active	:= (HMI_PAM_1._427 = 0) AND FALSE; //NOT USED AT THE MOMENT
	ALR[7177].Active	:= (HMI_PAM_1._431 = 0) AND (CFG_Par.FCI.Filltec OR CFG_Par.FCI.FTSystem OR CFG_Par.FCI.Heuft OR CFG_Par.FCI.Pressco OR CFG_Par.FCI.SIS OR CFG_Par.FCI.Stratec); //v999hema
	ALR[7178].Active	:= (HMI_PAM_1._435 = 0) AND CFG_Par.FCI.Heuft OR CFG_Par.FCI.Stratec;
	ALR[7179].Active	:= (HMI_PAM_1._439 = 0) AND CFG_Par.Doser.Present;

	ALR[7180].Active	:= NOT MC_InputOutput.Network.Filler.Status.FillerAbsolutePositionValid
							OR (NOT MC_InputOutput.Network.Filler.Status.RinserAbsolutePositionValid AND CFG_Par.Rinser.Present);
	//							OR (NOT MC_InputOutput.Network.Filler.Status.CapperAbsolutePositionValid AND CFG_Par.Lifting.Movements.Capper.UncouplingRequest) to be defined //V4.A.A.1.7.0
	//							OR (NOT MC_InputOutput.Network.Filler.Status.CrownerAbsolutePositionValid AND CFG_Par.Lifting.Movements.Crowner.UncouplingRequest);//V4.A.A.1.7.0

	//v4 200.2.0 eliminata logica
	ALR[7159].Active := MC_InputOutput.Network.Machine.Exceptions.FaultCamGeneration;//V.1.7.2
	// v4 200.2.0 eliminate logiche combi
END_ACTION

ACTION MNM_MotionAlarm:
	ALR[7002].Active	:= MC_InputOutput.Network.Machine.Exceptions.Fault;							//Motion -Motion Fault
	ALR[7004].Active	:= MC_InputOutput.Network.Machine.Exceptions.DcBusLowMachineException;		//Motion -DcBus voltage too low
	ALR[7005].Active	:= MC_InputOutput.Network.Machine.Exceptions.ExcessiveVelocityException;	//Motion -Excessive velocity requested
	ALR[7006].Active	:= MC_InputOutput.Network.Machine.Exceptions.ExcessiveAccException;			//Motion -Excessive acceleration requested
	ALR[7007].Active	:= MC_InputOutput.Network.Machine.Exceptions.NoAxisEnabledException;		//Motion -No Axis Enabled
	ALR[7008].Active	:= MC_InputOutput.Network.Machine.Exceptions.HomingException;				//Motion -Machine not in home
	ALR[7009].Active	:= MC_InputOutput.Network.Machine.Exceptions.BleederException;				//Motion -Bleeder error
	ALR[7013].Active	:= MC_InputOutput.Network.Machine.Exceptions.HmiChecksumException;			//Motion -HMI Checksum Error
	ALR[7014].Active	:= MC_InputOutput.Network.Machine.Exceptions.KochModuleNotReady;			//Motion -Koch Module Not ready

	IF (FillerFanIn1.OUT_Alarm		OR FillerFanIn2.OUT_Alarm		OR FillerFanIn3.OUT_Alarm		OR
		FillerFanIn4.OUT_Alarm		OR FillerFanIn5.OUT_Alarm		OR FillerFanIn6.OUT_Alarm		OR
		FillerFanIn7.OUT_Alarm		OR FillerFanIn8.OUT_Alarm		OR FillerFanIn9.OUT_Alarm		OR
		FillerFanIn10.OUT_Alarm		OR FillerFanMain.OUT_Alarm		OR FillerFanOut1.OUT_Alarm		OR
		FillerFanOut2.OUT_Alarm		OR FillerFanOut3.OUT_Alarm		OR FillerFanOut4.OUT_Alarm		OR
		FillerFanOut5.OUT_Alarm)	OR
		(OutletFanIn1.OUT_Alarm		OR OutletFanIn2.OUT_Alarm		OR OutletFanIn3.OUT_Alarm		OR
		OutletFanIn4.OUT_Alarm		OR OutletFanMain.OUT_Alarm		OR OutletFanOut1.OUT_Alarm		OR
		OutletFanOut2.OUT_Alarm		OR OutletFanOut3.OUT_Alarm		OR OutletFanOut4.OUT_Alarm)		OR
		MC_InputOutput.Network.Machine.Exceptions.FanSeamearFault THEN
		ALR[7015].Active := TRUE;	//Motion -Servoventilation Drive Error
	ELSE
		ALR[7015].Active := FALSE;	//Motion -Servoventilation Drive Error
	END_IF

	IF TMR_TON_TimeoutModality.Q THEN
		ALR[7016].Active	:= TRUE;
	ELSIF AID.DataOut.Reset THEN
		ALR[7016].Active	:= FALSE;
	END_IF

END_ACTION

ACTION MNM_MotionModuleAlarm:
	(*MASTER MODULE *)
	ALR[7470].Active	:= MC_InputOutput.Network.Machine.Status.ModuleNotInitialized;//1.7.2a
	(* FILLER MODULE *)
	ALR[7199].Active	:= MC_InputOutput.Network.Filler.Status.ModuleNotInitialized;			//Motion -Filler module not initialized

	IF NOT MC_InputOutput.Network.Filler.Status.ModuleNotInitialized THEN
		ALR[7200].Active	:= MC_InputOutput.Network.Filler.Exceptions.CarouselTrackException;		//Motion -Filler Carousel: Lag error
		ALR[7201].Active	:= MC_InputOutput.Network.Filler.Exceptions.CarouselHomeException;		//Motion -Filler Carousel: Not homed
		ALR[7202].Active	:= MC_InputOutput.Network.Filler.Exceptions.CarouselTorqueException;	//Motion -Filler Carousel: Torque limit exceeded
		ALR[7203].Active	:= MC_InputOutput.Network.Filler.Exceptions.CarouselDriveException;		//Motion -Filler Carousel: Drive error
		ALR[7204].Active	:= MC_InputOutput.Network.Filler.Exceptions.CarouselSafetyException;	//Motion -Filler Carousel: Safety violation
		ALR[7205].Active	:= MC_InputOutput.Network.Filler.Exceptions.CarouselNotInOpException;	//Motion -Filler Carousel: Not in operation

		ALR[7206].Active	:= MC_InputOutput.Network.Filler.Exceptions.Inlet01TrackException;		//Motion -Filler Inlet: Lag error
		ALR[7207].Active	:= MC_InputOutput.Network.Filler.Exceptions.Inlet01HomeException;		//Motion -Filler Inlet: Not homed
		ALR[7208].Active	:= MC_InputOutput.Network.Filler.Exceptions.Inlet01TorqueException;		//Motion -Filler Inlet: Torque limit exceeded
		ALR[7209].Active	:= MC_InputOutput.Network.Filler.Exceptions.Inlet01DriveException;		//Motion -Filler Inlet: Drive error
		ALR[7210].Active	:= MC_InputOutput.Network.Filler.Exceptions.Inlet01SafetyException;		//Motion -Filler Inlet: Safety violation
		ALR[7211].Active	:= MC_InputOutput.Network.Filler.Exceptions.Inlet01NotInOpException;	//Motion -Filler Inlet: Not in operation

		ALR[7212].Active	:= MC_InputOutput.Network.Filler.Exceptions.Inlet02TrackException;		//Motion -Filler Inlet: Lag error
		ALR[7213].Active	:= MC_InputOutput.Network.Filler.Exceptions.Inlet02HomeException;		//Motion -Filler Inlet: Not homed
		ALR[7214].Active	:= MC_InputOutput.Network.Filler.Exceptions.Inlet02TorqueException;		//Motion -Filler Inlet: Torque limit exceeded
		ALR[7215].Active	:= MC_InputOutput.Network.Filler.Exceptions.Inlet02DriveException;		//Motion -Filler Inlet: Drive error
		ALR[7216].Active	:= MC_InputOutput.Network.Filler.Exceptions.Inlet02SafetyException;		//Motion -Filler Inlet: Safety violation
		ALR[7217].Active	:= MC_InputOutput.Network.Filler.Exceptions.Inlet02NotInOpException;	//Motion -Filler Inlet: Not in operation

		ALR[7218].Active	:= MC_InputOutput.Network.Filler.Exceptions.Inlet03TrackException;		//Motion -Filler Inlet: Lag error
		ALR[7219].Active	:= MC_InputOutput.Network.Filler.Exceptions.Inlet03HomeException;		//Motion -Filler Inlet: Not homed
		ALR[7220].Active	:= MC_InputOutput.Network.Filler.Exceptions.Inlet03TorqueException;		//Motion -Filler Inlet: Torque limit exceeded
		ALR[7221].Active	:= MC_InputOutput.Network.Filler.Exceptions.Inlet03DriveException;		//Motion -Filler Inlet: Drive error
		ALR[7222].Active	:= MC_InputOutput.Network.Filler.Exceptions.Inlet03SafetyException;		//Motion -Filler Inlet: Safety violation
		ALR[7223].Active	:= MC_InputOutput.Network.Filler.Exceptions.Inlet03NotInOpException;	//Motion -Filler Inlet: Not in operation

		ALR[7224].Active	:= MC_InputOutput.Network.Filler.Exceptions.Inlet04TrackException;		//Motion -Filler Inlet: Lag error
		ALR[7225].Active	:= MC_InputOutput.Network.Filler.Exceptions.Inlet04HomeException;		//Motion -Filler Inlet: Not homed
		ALR[7226].Active	:= MC_InputOutput.Network.Filler.Exceptions.Inlet04TorqueException;		//Motion -Filler Inlet: Torque limit exceeded
		ALR[7227].Active	:= MC_InputOutput.Network.Filler.Exceptions.Inlet04DriveException;		//Motion -Filler Inlet: Drive error
		ALR[7228].Active	:= MC_InputOutput.Network.Filler.Exceptions.Inlet04SafetyException;		//Motion -Filler Inlet: Safety violation
		ALR[7229].Active	:= MC_InputOutput.Network.Filler.Exceptions.Inlet04NotInOpException;	//Motion -Filler Inlet: Not in operation

		ALR[7230].Active	:= MC_InputOutput.Network.Filler.Exceptions.Inlet05TrackException;		//Motion -Filler Inlet: Lag error
		ALR[7231].Active	:= MC_InputOutput.Network.Filler.Exceptions.Inlet05HomeException;		//Motion -Filler Inlet: Not homed
		ALR[7232].Active	:= MC_InputOutput.Network.Filler.Exceptions.Inlet05TorqueException;		//Motion -Filler Inlet: Torque limit exceeded
		ALR[7233].Active	:= MC_InputOutput.Network.Filler.Exceptions.Inlet05DriveException;		//Motion -Filler Inlet: Drive error
		ALR[7234].Active	:= MC_InputOutput.Network.Filler.Exceptions.Inlet05SafetyException;		//Motion -Filler Inlet: Safety violation
		ALR[7235].Active	:= MC_InputOutput.Network.Filler.Exceptions.Inlet05NotInOpException;	//Motion -Filler Inlet: Not in operation

		ALR[7236].Active	:= MC_InputOutput.Network.Filler.Exceptions.Inlet06TrackException;		//Motion -Filler Inlet: Lag error
		ALR[7237].Active	:= MC_InputOutput.Network.Filler.Exceptions.Inlet06HomeException;		//Motion -Filler Inlet: Not homed
		ALR[7238].Active	:= MC_InputOutput.Network.Filler.Exceptions.Inlet06TorqueException;		//Motion -Filler Inlet: Torque limit exceeded
		ALR[7239].Active	:= MC_InputOutput.Network.Filler.Exceptions.Inlet06DriveException;		//Motion -Filler Inlet: Drive error
		ALR[7240].Active	:= MC_InputOutput.Network.Filler.Exceptions.Inlet06SafetyException;		//Motion -Filler Inlet: Safety violation
		ALR[7241].Active	:= MC_InputOutput.Network.Filler.Exceptions.Inlet06NotInOpException;	//Motion -Filler Inlet: Not in operation

		ALR[7242].Active	:= MC_InputOutput.Network.Filler.Exceptions.Inlet07TrackException;		//Motion -Filler Inlet: Lag error
		ALR[7243].Active	:= MC_InputOutput.Network.Filler.Exceptions.Inlet07HomeException;		//Motion -Filler Inlet: Not homed
		ALR[7244].Active	:= MC_InputOutput.Network.Filler.Exceptions.Inlet07TorqueException;		//Motion -Filler Inlet: Torque limit exceeded
		ALR[7245].Active	:= MC_InputOutput.Network.Filler.Exceptions.Inlet07DriveException;		//Motion -Filler Inlet: Drive error
		ALR[7246].Active	:= MC_InputOutput.Network.Filler.Exceptions.Inlet07SafetyException;		//Motion -Filler Inlet: Safety violation
		ALR[7247].Active	:= MC_InputOutput.Network.Filler.Exceptions.Inlet07NotInOpException;	//Motion -Filler Inlet: Not in operation

		ALR[7248].Active	:= MC_InputOutput.Network.Filler.Exceptions.Inlet08TrackException;		//Motion -Filler Inlet: Lag error
		ALR[7249].Active	:= MC_InputOutput.Network.Filler.Exceptions.Inlet08HomeException;		//Motion -Filler Inlet: Not homed
		ALR[7250].Active	:= MC_InputOutput.Network.Filler.Exceptions.Inlet08TorqueException;		//Motion -Filler Inlet: Torque limit exceeded
		ALR[7251].Active	:= MC_InputOutput.Network.Filler.Exceptions.Inlet08DriveException;		//Motion -Filler Inlet: Drive error
		ALR[7252].Active	:= MC_InputOutput.Network.Filler.Exceptions.Inlet08SafetyException;		//Motion -Filler Inlet: Safety violation
		ALR[7253].Active	:= MC_InputOutput.Network.Filler.Exceptions.Inlet08NotInOpException;	//Motion -Filler Inlet: Not in operation

		ALR[7254].Active	:= MC_InputOutput.Network.Filler.Exceptions.Inlet09TrackException;		//Motion -Filler Inlet: Lag error
		ALR[7255].Active	:= MC_InputOutput.Network.Filler.Exceptions.Inlet09HomeException;		//Motion -Filler Inlet: Not homed
		ALR[7256].Active	:= MC_InputOutput.Network.Filler.Exceptions.Inlet09TorqueException;		//Motion -Filler Inlet: Torque limit exceeded
		ALR[7257].Active	:= MC_InputOutput.Network.Filler.Exceptions.Inlet09DriveException;		//Motion -Filler Inlet: Drive error
		ALR[7258].Active	:= MC_InputOutput.Network.Filler.Exceptions.Inlet09SafetyException;		//Motion -Filler Inlet: Safety violation
		ALR[7259].Active	:= MC_InputOutput.Network.Filler.Exceptions.Inlet09NotInOpException;	//Motion -Filler Inlet: Not in operation

		ALR[7260].Active	:= MC_InputOutput.Network.Filler.Exceptions.Inlet10TrackException;		//Motion -Filler Inlet: Lag error
		ALR[7261].Active	:= MC_InputOutput.Network.Filler.Exceptions.Inlet10HomeException;		//Motion -Filler Inlet: Not homed
		ALR[7262].Active	:= MC_InputOutput.Network.Filler.Exceptions.Inlet10TorqueException;		//Motion -Filler Inlet: Torque limit exceeded
		ALR[7263].Active	:= MC_InputOutput.Network.Filler.Exceptions.Inlet10DriveException;		//Motion -Filler Inlet: Drive error
		ALR[7264].Active	:= MC_InputOutput.Network.Filler.Exceptions.Inlet10SafetyException;		//Motion -Filler Inlet: Safety violation
		ALR[7265].Active	:= MC_InputOutput.Network.Filler.Exceptions.Inlet10NotInOpException;	//Motion -Filler Inlet: Not in operation

		ALR[7266].Active	:= MC_InputOutput.Network.Filler.Exceptions.Outlet01TrackException;		//Motion -Filler Outlet: Lag error
		ALR[7267].Active	:= MC_InputOutput.Network.Filler.Exceptions.Outlet01HomeException;		//Motion -Filler Outlet: Not homed
		ALR[7268].Active	:= MC_InputOutput.Network.Filler.Exceptions.Outlet01TorqueException;	//Motion -Filler Outlet: Torque limit exceeded
		ALR[7269].Active	:= MC_InputOutput.Network.Filler.Exceptions.Outlet01DriveException;		//Motion -Filler Outlet: Drive error
		ALR[7270].Active	:= MC_InputOutput.Network.Filler.Exceptions.Outlet01SafetyException;	//Motion -Filler Outlet: Safety violation
		ALR[7271].Active	:= MC_InputOutput.Network.Filler.Exceptions.Outlet01NotInOpException;	//Motion -Filler Outlet: Not in operation

		ALR[7272].Active	:= MC_InputOutput.Network.Filler.Exceptions.Outlet02TrackException;		//Motion -Filler Outlet: Lag error
		ALR[7273].Active	:= MC_InputOutput.Network.Filler.Exceptions.Outlet02HomeException;		//Motion -Filler Outlet: Not homed
		ALR[7274].Active	:= MC_InputOutput.Network.Filler.Exceptions.Outlet02TorqueException;	//Motion -Filler Outlet: Torque limit exceeded
		ALR[7275].Active	:= MC_InputOutput.Network.Filler.Exceptions.Outlet02DriveException;		//Motion -Filler Outlet: Drive error
		ALR[7276].Active	:= MC_InputOutput.Network.Filler.Exceptions.Outlet02SafetyException;	//Motion -Filler Outlet: Safety violation
		ALR[7277].Active	:= MC_InputOutput.Network.Filler.Exceptions.Outlet02NotInOpException;	//Motion -Filler Outlet: Not in operation

		ALR[7278].Active	:= MC_InputOutput.Network.Filler.Exceptions.Outlet03TrackException;		//Motion -Filler Outlet: Lag error
		ALR[7279].Active	:= MC_InputOutput.Network.Filler.Exceptions.Outlet03HomeException;		//Motion -Filler Outlet: Not homed
		ALR[7280].Active	:= MC_InputOutput.Network.Filler.Exceptions.Outlet03TorqueException;	//Motion -Filler Outlet: Torque limit exceeded
		ALR[7281].Active	:= MC_InputOutput.Network.Filler.Exceptions.Outlet03DriveException;		//Motion -Filler Outlet: Drive error
		ALR[7282].Active	:= MC_InputOutput.Network.Filler.Exceptions.Outlet03SafetyException;	//Motion -Filler Outlet: Safety violation
		ALR[7283].Active	:= MC_InputOutput.Network.Filler.Exceptions.Outlet03NotInOpException;	//Motion -Filler Outlet: Not in operation
	ELSIF EDGEPOS(MC_InputOutput.Network.Filler.Status.ModuleNotInitialized) THEN
		FOR VAR_i := 7200 TO 7283 DO
			ALR[VAR_i].Active := FALSE;
		END_FOR
	END_IF

	(* INLET MODULE *)
	ALR[7049].Active	:= MC_InputOutput.Network.Inlet.Status.ModuleNotInitialized;			//Motion -Inlet module not initialized

	IF NOT MC_InputOutput.Network.Inlet.Status.ModuleNotInitialized THEN
		ALR[7050].Active	:= MC_InputOutput.Network.Inlet.Exceptions.MainAxisTrackException;		//Motion -Inlet Carousel: Lag error
		ALR[7051].Active	:= MC_InputOutput.Network.Inlet.Exceptions.MainAxisHomeException;		//Motion -Inlet Carousel: Not homed
		ALR[7052].Active	:= MC_InputOutput.Network.Inlet.Exceptions.MainAxisTorqueException;		//Motion -Inlet Carousel: Torque limit exceeded
		ALR[7053].Active	:= MC_InputOutput.Network.Inlet.Exceptions.MainAxisDriveException;		//Motion -Inlet Carousel: Drive error
		ALR[7054].Active	:= MC_InputOutput.Network.Inlet.Exceptions.MainAxisSafetyException;		//Motion -Inlet Carousel: Safety violation
		ALR[7055].Active	:= MC_InputOutput.Network.Inlet.Exceptions.MainAxisNotInOpException;	//Motion -Inlet Carousel: Not in operation
	ELSIF EDGEPOS(MC_InputOutput.Network.Inlet.Status.ModuleNotInitialized) THEN
		FOR VAR_i := 7050 TO 7055 DO
			ALR[VAR_i].Active := FALSE;
		END_FOR
	END_IF

	(* OUTLET MODULE *)
	ALR[7349].Active	:= MC_InputOutput.Network.Outlet.Status.ModuleNotInitialized;			//Motion -Seamer module not initialized

	IF NOT MC_InputOutput.Network.Outlet.Status.ModuleNotInitialized THEN
		ALR[7350].Active	:= MC_InputOutput.Network.Outlet.Exceptions.MainAxisTrackException;		//Motion -Seamer Carousel: Lag error
		ALR[7351].Active	:= MC_InputOutput.Network.Outlet.Exceptions.MainAxisHomeException;		//Motion -Seamer Carousel: Not homed
		ALR[7352].Active	:= MC_InputOutput.Network.Outlet.Exceptions.MainAxisTorqueException;	//Motion -Seamer Carousel: Torque limit exceeded
		ALR[7353].Active	:= MC_InputOutput.Network.Outlet.Exceptions.MainAxisDriveException;		//Motion -Seamer Carousel: Drive error
		ALR[7354].Active	:= MC_InputOutput.Network.Outlet.Exceptions.MainAxisSafetyException;	//Motion -Seamer Carousel: Safety violation
		ALR[7355].Active	:= MC_InputOutput.Network.Outlet.Exceptions.MainAxisNotInOpException;	//Motion -Seamer Carousel: Not in operation

		ALR[7416].Active	:= MC_InputOutput.Network.Outlet.Exceptions.Outlet01TrackException;		//Motion -Seamer Carousel: Lag error
		ALR[7417].Active	:= MC_InputOutput.Network.Outlet.Exceptions.Outlet01HomeException;		//Motion -Seamer Carousel: Not homed
		ALR[7418].Active	:= MC_InputOutput.Network.Outlet.Exceptions.Outlet01TorqueException;	//Motion -Seamer Carousel: Torque limit exceeded
		ALR[7419].Active	:= MC_InputOutput.Network.Outlet.Exceptions.Outlet01DriveException;		//Motion -Seamer Carousel: Drive error
		ALR[7420].Active	:= MC_InputOutput.Network.Outlet.Exceptions.Outlet01SafetyException;	//Motion -Seamer Carousel: Safety violation
		ALR[7421].Active	:= MC_InputOutput.Network.Outlet.Exceptions.Outlet01NotInOpException;	//Motion -Seamer Carousel: Not in operation
	ELSIF EDGEPOS(MC_InputOutput.Network.Outlet.Status.ModuleNotInitialized) THEN
		FOR VAR_i := 7350 TO 7421 DO
			ALR[VAR_i].Active := FALSE;
		END_FOR
	END_IF
END_ACTION
```

#### MNM_DisableMotorManagement.st
```iecst
ACTION MNM_DisableMotorManagement:
 // in wait riabilito tutto ipotesi uno
	VAR_MNM_DefaultAxisConfig := DOS.DataOut.AllAxisEnableRequest OR (TNK.DataOut.DummyContainersDis AND TNK.DataOut.CipMode);

	IF DOS.DataOut.AxisEnableRequest AND VAR_MNM_AxisDisableStep <> 1 AND NOT DOS.DataOut.RunOnlyHemaAxisRequest THEN
		VAR_MNM_AxisDisableStep := 1;
	ELSIF DOS.DataOut.AxisDisableRequest AND VAR_MNM_AxisDisableStep <> 2 THEN
		VAR_MNM_AxisDisableStep := 2;
	ELSIF DOS.DataOut.RunOnlyHemaAxisRequest AND VAR_MNM_AxisDisableStep <> 3 THEN
		VAR_MNM_AxisDisableStep := 3;
	ELSIF DOS.DataOut.RunRinserHemaAxisRequest AND VAR_MNM_AxisDisableStep <> 4 THEN
		VAR_MNM_AxisDisableStep := 4;
	ELSIF RNS.DataOut.RunOnlyRinserAxisRequest AND VAR_MNM_AxisDisableStep <> 5 THEN
		VAR_MNM_AxisDisableStep := 5;
	ELSIF VAR_MNM_DefaultAxisConfig AND VAR_MNM_AxisDisableStep <> 0 THEN
		VAR_MNM_AxisDisableStep := 0;
	END_IF

	IF VAR_MNM_AxisConfigLoadedNumber <> VAR_MNM_AxisDisableStep OR ALR[3015].Active OR ALR[3016].Active  THEN
		VAR_MNM_NormalStop := TRUE;
	ELSIF VAR_MNM_AxisConfigLoadedNumber = VAR_MNM_AxisDisableStep THEN
		VAR_MNM_NormalStop := FALSE;
	END_IF

	CASE VAR_MNM_AxisDisableStep OF

		0: // Configuration of Motor must be disabled //Default Motor Configuration all axis are Enabled
			IF NOT MNM.DataOut.MachineRunning THEN
				memcpy( ADR(MC_InputOutput.Network.Filler.Commands.MotorDisableIndex),ADR(CFG_MC.MotorDisableConfig[0]), SIZEOF(CFG_MC.MotorDisableConfig[0]));
			END_IF
			MNM.DataOut.ConfigReqLoaded := (memcmp( ADR( MC_InputOutput.Network.Filler.Status.AxisDisabledFeedBack), ADR(CFG_MC.MotorDisableConfig[0]) ,SIZEOF(CFG_MC.MotorDisableConfig[0])) = 0);

			IF 	MNM.DataOut.ConfigReqLoaded THEN
				MNM.DataOut.ConfigReqLoaded	:= FALSE;
				VAR_MNM_AxisConfigLoadedNumber	:= 0;
			END_IF

		1:// configuration 1 request to MC , wait answer from MC program //DOSER ENABLE
			IF NOT MNM.DataOut.MachineRunning THEN
				memcpy( ADR(MC_InputOutput.Network.Filler.Commands.MotorDisableIndex),ADR(CFG_MC.MotorDisableConfig[1]), SIZEOF(CFG_MC.MotorDisableConfig[1]));
			END_IF
			MNM.DataOut.ConfigReqLoaded := (memcmp( ADR( MC_InputOutput.Network.Filler.Status.AxisDisabledFeedBack), ADR(CFG_MC.MotorDisableConfig[1]) ,SIZEOF(CFG_MC.MotorDisableConfig[1])) = 0);

			IF 	MNM.DataOut.ConfigReqLoaded AND NOT DOS.DataOut.AxisEnableRequest THEN
				MNM.DataOut.ConfigReqLoaded	:= FALSE;
				VAR_MNM_AxisConfigLoadedNumber	:= 1;
			END_IF
		2:// configuration 1 request to MC , wait answer from MC program DOSER DISABLE
			IF NOT MNM.DataOut.MachineRunning THEN
				memcpy( ADR(MC_InputOutput.Network.Filler.Commands.MotorDisableIndex),ADR(CFG_MC.MotorDisableConfig[2]), SIZEOF(CFG_MC.MotorDisableConfig[2]));
			 END_IF
			MNM.DataOut.ConfigReqLoaded := (memcmp( ADR( MC_InputOutput.Network.Filler.Status.AxisDisabledFeedBack), ADR(CFG_MC.MotorDisableConfig[2]) ,SIZEOF(CFG_MC.MotorDisableConfig[2])) = 0);

			IF 	MNM.DataOut.ConfigReqLoaded AND NOT DOS.DataOut.AxisDisableRequest THEN
				MNM.DataOut.ConfigReqLoaded	:= FALSE;
				VAR_MNM_AxisConfigLoadedNumber	:= 2;
			END_IF

		3:// configuration 1 request to MC , wait answer from MC program DOSER ONLY
			IF NOT MNM.DataOut.MachineRunning THEN
				memcpy( ADR(MC_InputOutput.Network.Filler.Commands.MotorDisableIndex),ADR(CFG_MC.MotorDisableConfig[3]), SIZEOF(CFG_MC.MotorDisableConfig[3]));
			END_IF
			MNM.DataOut.ConfigReqLoaded := (memcmp( ADR( MC_InputOutput.Network.Filler.Status.AxisDisabledFeedBack), ADR(CFG_MC.MotorDisableConfig[3]) ,SIZEOF(CFG_MC.MotorDisableConfig[3])) = 0);

			IF MNM.DataOut.ConfigReqLoaded THEN
				VAR_MNM_AxisConfigLoadedNumber	:= 3;
			END_IF

			IF 	MNM.DataOut.ConfigReqLoaded AND NOT DOS.DataOut.RunOnlyHemaAxisRequest THEN
				MNM.DataOut.ConfigReqLoaded	:= FALSE;
				VAR_MNM_AxisConfigLoadedNumber	:= 3;
			END_IF

		4:// configuration 1 request to MC , wait answer from MC program DOSER + RINSER ONLY
			IF NOT MNM.DataOut.MachineRunning THEN
				memcpy( ADR(MC_InputOutput.Network.Filler.Commands.MotorDisableIndex),ADR(CFG_MC.MotorDisableConfig[4]), SIZEOF(CFG_MC.MotorDisableConfig[4]));
			END_IF
			MNM.DataOut.ConfigReqLoaded := (memcmp( ADR( MC_InputOutput.Network.Filler.Status.AxisDisabledFeedBack), ADR(CFG_MC.MotorDisableConfig[4]) ,SIZEOF(CFG_MC.MotorDisableConfig[4])) = 0);

			IF MNM.DataOut.ConfigReqLoaded THEN
				VAR_MNM_AxisConfigLoadedNumber	:= 4;
			END_IF

			IF 	MNM.DataOut.ConfigReqLoaded AND NOT DOS.DataOut.RunRinserHemaAxisRequest THEN
				MNM.DataOut.ConfigReqLoaded	:= FALSE;
				VAR_MNM_AxisConfigLoadedNumber	:= 4;
			END_IF
		5:// configuration 1 request to MC , wait answer from MC program RINSER ONLY
			IF NOT MNM.DataOut.MachineRunning THEN
				memcpy( ADR(MC_InputOutput.Network.Filler.Commands.MotorDisableIndex),ADR(CFG_MC.MotorDisableConfig[5]), SIZEOF(CFG_MC.MotorDisableConfig[5]));
			END_IF
			MNM.DataOut.ConfigReqLoaded := (memcmp( ADR( MC_InputOutput.Network.Filler.Status.AxisDisabledFeedBack), ADR(CFG_MC.MotorDisableConfig[5]) ,SIZEOF(CFG_MC.MotorDisableConfig[5])) = 0);

			IF 	MNM.DataOut.ConfigReqLoaded AND NOT RNS.DataOut.RunOnlyRinserAxisRequest THEN
				MNM.DataOut.ConfigReqLoaded	:= FALSE;
				VAR_MNM_AxisConfigLoadedNumber	:= 5;
			END_IF
	END_CASE
END_ACTION
```

#### MNM_MachineSpeedManagemant.st
```iecst
ACTION MNM_MachineSpeedManagemant:
	VAR_ModuleSpeed.Machine	:= 0.0;
	VAR_ModuleSpeed.Inlet	:= 0.0;
	VAR_ModuleSpeed.Filler	:= 0.0;
	VAR_ModuleSpeed.Outlet	:= 0.0;

	VAR_FixSpeedActive		:= 0;
	VAR_InFixSpeedActive	:= 0;
	VAR_FlrFixSpeedActive	:= 0;
	VAR_OutFixSpeedActive	:= 0;

	IF NOT MC_InputOutput.Network.Machine.Status.MultiModalityActive THEN
		FOR iSpeed := 1 TO CST_FixSpeedMax DO
			IF VAR_FixSpeed[iSpeed].Req AND VAR_FixSpeedActive = 0 THEN
				VAR_ModuleSpeed.Machine		:= VAR_FixSpeed[iSpeed].Value;
				VAR_FixSpeedActive			:= iSpeed;
			END_IF

			IF VAR_FixSpeedActive <> 0 AND VAR_FixSpeed[iSpeed].Req THEN
				IF VAR_FixSpeed[VAR_FixSpeedActive].Interruptible THEN
					VAR_ModuleSpeed.Machine		:= VAR_FixSpeed[iSpeed].Value;
					VAR_FixSpeedActive			:= iSpeed;
				END_IF
			END_IF

			TON_ReachedDelay[iSpeed](
			IN := FC_SpeedCheck(IN_SpeedReq := VAR_FixSpeed[iSpeed].Value, IN_SpeedAct := MC_InputOutput.Network.Machine.Status.ActualSpeed, IN_Mode := VAR_FixSpeed[iSpeed].CmpMode),
			PT := t#2s
			);
			VAR_FixSpeed[iSpeed].Reached := TON_ReachedDelay[iSpeed].Q AND VAR_FixSpeed[iSpeed].Req;
		END_FOR
	ELSE
		FOR iSpeed := 1 TO CST_FixSpeedMax DO
			IF VAR_FixSpeed[iSpeed].Req AND VAR_FixSpeedActive = 0 THEN//1.7.2
				IF VAR_FixSpeed[iSpeed].Module = 1 THEN
					VAR_ModuleSpeed.Inlet	:= VAR_FixSpeed[iSpeed].Value;
					VAR_InFixSpeedActive	:= iSpeed;
				ELSIF VAR_FixSpeed[iSpeed].Module = 2 THEN
					VAR_ModuleSpeed.Filler	:= VAR_FixSpeed[iSpeed].Value;
					VAR_FlrFixSpeedActive	:= iSpeed;
				ELSIF VAR_FixSpeed[iSpeed].Module = 3 THEN
					VAR_ModuleSpeed.Outlet	:= VAR_FixSpeed[iSpeed].Value;
					VAR_OutFixSpeedActive	:= iSpeed;
				ELSIF VAR_FixSpeed[iSpeed].Module = 9 THEN
					VAR_ModuleSpeed.Inlet	:= VAR_FixSpeed[iSpeed].Value;
					VAR_ModuleSpeed.Filler	:= VAR_FixSpeed[iSpeed].Value;
					VAR_ModuleSpeed.Outlet	:= VAR_FixSpeed[iSpeed].Value;
					VAR_InFixSpeedActive	:= iSpeed;
					VAR_FlrFixSpeedActive	:= iSpeed;
					VAR_OutFixSpeedActive	:= iSpeed;
				END_IF
			END_IF

			IF VAR_InFixSpeedActive <> 0 AND VAR_FixSpeed[iSpeed].Req AND VAR_FixSpeed[iSpeed].Module = 1 THEN
				IF VAR_FixSpeed[VAR_InFixSpeedActive].Interruptible THEN
					VAR_ModuleSpeed.Inlet	:= VAR_FixSpeed[iSpeed].Value;
					VAR_InFixSpeedActive	:= iSpeed;
				END_IF
			END_IF

			IF VAR_FlrFixSpeedActive <> 0 AND VAR_FixSpeed[iSpeed].Req AND VAR_FixSpeed[iSpeed].Module = 2 THEN
				IF VAR_FixSpeed[VAR_FlrFixSpeedActive].Interruptible THEN
					VAR_ModuleSpeed.Filler	:= VAR_FixSpeed[iSpeed].Value;
					VAR_FlrFixSpeedActive	:= iSpeed;
				END_IF
			END_IF

			IF VAR_OutFixSpeedActive <> 0 AND VAR_FixSpeed[iSpeed].Req AND VAR_FixSpeed[iSpeed].Module = 3 THEN
				IF VAR_FixSpeed[VAR_OutFixSpeedActive].Interruptible THEN
					VAR_ModuleSpeed.Outlet	:= VAR_FixSpeed[iSpeed].Value;
					VAR_OutFixSpeedActive	:= iSpeed;
				END_IF
			END_IF

			IF VAR_FixSpeed[iSpeed].Module = 1 THEN
				TON_ReachedDelay[iSpeed](
				IN := FC_SpeedCheck(IN_SpeedReq := VAR_FixSpeed[iSpeed].Value, IN_SpeedAct := MC_InputOutput.Network.Inlet.Status.Velocity, IN_Mode := VAR_FixSpeed[iSpeed].CmpMode),
				PT := t#2s
				);
			END_IF

			IF VAR_FixSpeed[iSpeed].Module = 2 THEN
				TON_ReachedDelay[iSpeed](
				IN := FC_SpeedCheck(IN_SpeedReq := VAR_FixSpeed[iSpeed].Value, IN_SpeedAct := MC_InputOutput.Network.Filler.Status.Velocity, IN_Mode := VAR_FixSpeed[iSpeed].CmpMode),
				PT := t#2s
				);
			END_IF

			IF VAR_FixSpeed[iSpeed].Module = 3 THEN
				TON_ReachedDelay[iSpeed](
				IN := FC_SpeedCheck(IN_SpeedReq := VAR_FixSpeed[iSpeed].Value, IN_SpeedAct := MC_InputOutput.Network.Outlet.Status.Velocity, IN_Mode := VAR_FixSpeed[iSpeed].CmpMode),
				PT := t#2s
				);
			END_IF

			IF VAR_FixSpeed[iSpeed].Module = 9 THEN
				IF MC_InputOutput.Network.Inlet.Status.ModuleReal THEN
					TON_ReachedDelay[iSpeed].IN	:= FC_SpeedCheck(	IN_SpeedReq := VAR_FixSpeed[iSpeed].Value,
					IN_SpeedAct := MC_InputOutput.Network.Inlet.Status.Velocity,
					IN_Mode := VAR_FixSpeed[iSpeed].CmpMode);
				ELSE
					TON_ReachedDelay[iSpeed].IN := TRUE;
				END_IF

				IF MC_InputOutput.Network.Filler.Status.ModuleReal THEN
					TON_ReachedDelay[iSpeed].IN	:= FC_SpeedCheck(	IN_SpeedReq := VAR_FixSpeed[iSpeed].Value,
					IN_SpeedAct := MC_InputOutput.Network.Filler.Status.Velocity,
					IN_Mode := VAR_FixSpeed[iSpeed].CmpMode) AND TON_ReachedDelay[iSpeed].IN;
				ELSE
					TON_ReachedDelay[iSpeed].IN := TON_ReachedDelay[iSpeed].IN;
				END_IF

				IF MC_InputOutput.Network.Outlet.Status.ModuleReal THEN
					TON_ReachedDelay[iSpeed].IN	:= FC_SpeedCheck(	IN_SpeedReq := VAR_FixSpeed[iSpeed].Value,
					IN_SpeedAct := MC_InputOutput.Network.Outlet.Status.Velocity,
					IN_Mode := VAR_FixSpeed[iSpeed].CmpMode) AND TON_ReachedDelay[iSpeed].IN;
				ELSE
					TON_ReachedDelay[iSpeed].IN := TON_ReachedDelay[iSpeed].IN;
				END_IF

				TON_ReachedDelay[iSpeed](
				PT := t#2s
				);
			END_IF
			VAR_FixSpeed[iSpeed].Reached := TON_ReachedDelay[iSpeed].Q AND VAR_FixSpeed[iSpeed].Req;
		END_FOR
	END_IF

	IF VAR_FixSpeedActive = 0 THEN
		VAR_ModuleSpeed.Machine	:= DINT_TO_REAL(HMI_MNM_FlrSpeedWidget.AutoSpeedReq);
	END_IF

	IF VAR_InFixSpeedActive = 0 THEN
		VAR_ModuleSpeed.Inlet;
	END_IF

	IF VAR_FlrFixSpeedActive = 0 THEN
		VAR_ModuleSpeed.Filler	:= DINT_TO_REAL(HMI_MNM_FlrSpeedWidget.AutoSpeedReq);
	END_IF

	IF VAR_OutFixSpeedActive = 0 THEN
		VAR_ModuleSpeed.Outlet	:= DINT_TO_REAL(HMI_MNM_SmrSpeedWidget.AutoSpeedReq);
	END_IF

	IF VAR_FixSpeedActive <> 0 OR VAR_InFixSpeedActive <> 0 OR VAR_FlrFixSpeedActive <> 0 OR VAR_OutFixSpeedActive <> 0 THEN
		VAR_MNM_FixSpeedReq := TRUE;
	ELSE
		VAR_MNM_FixSpeedReq := FALSE;
	END_IF

END_ACTION
```

### Package Logical/08_RNS - Rinser: gestione Sciacquatrice

### Program Logical/08_RNS/RNS (IEC) - RNS Main Program - C#4 - 100ms

#### RNS.sfc - Cyclic code
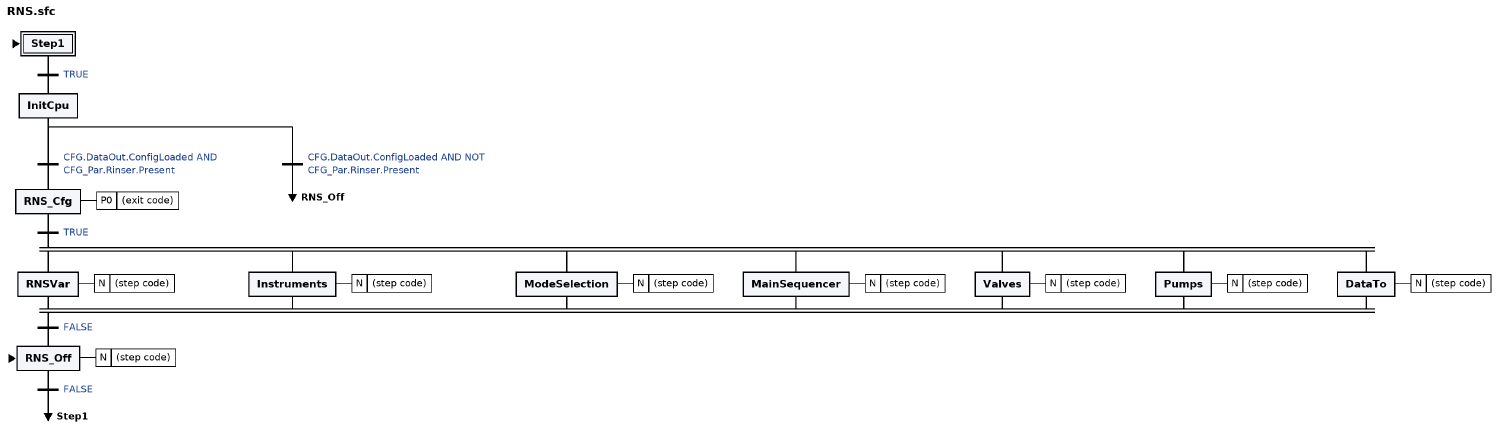
```iecst
PROGRAM _CYCLIC
INITIAL_STEP Step1:
END_STEP
TRANSITION FROM Step1 TO InitCpu:=
TRUE
END_TRANSITION
STEP InitCpu:
END_STEP
TRANSITION PRESENT FROM InitCpu TO RNS_Cfg:=
CFG.DataOut.ConfigLoaded AND CFG_Par.Rinser.Present
END_TRANSITION
TRANSITION NOT PRESENT FROM InitCpu TO RNS_Off:=
CFG.DataOut.ConfigLoaded AND NOT CFG_Par.Rinser.Present
END_TRANSITION
(* @SFCISJUMP := 'RNS_Off' *)
STEP RNS_Cfg:
END_STEP
EXIT_ACTION
RNS_Hardware_CFG;

HMI_CFG_PAC_1._201	:= TRUE;
HMI_CFG_PAC_1._202	:= TRUE;

HMI_CFG_PAM_1._014 	:= CFG_Par.Rinser.PressureNozzleControlInsertion;
HMI_CFG_PAM_1._015 	:= CFG_Par.Rinser.PressureNozzleControlContinous;
HMI_CFG_PAM_1._081 	:= CFG_Par.Rinser.PressureNozzleControlInsertion;
HMI_CFG_PAM_1._083 	:= CFG_Par.Rinser.PressureNozzleControlContinous;
HMI_CFG_PAM_1._085 	:= CFG_Par.Rinser.PressureNozzleControlContinous;
HMI_CFG_PAM_1._087 	:= CFG_Par.Rinser.PressureNozzleControlInsertion;
HMI_CFG_PAM_1._089 	:= CFG_Par.Rinser.PressureNozzleControlContinous;
HMI_CFG_PAM_1._090 	:= CFG_Par.Rinser.PressureNozzleControlInsertion;
HMI_CFG_PAM_1._091 	:= CFG_Par.Rinser.PressureNozzleControlContinous;
//RVB202 SP
HMI_CFG_PAM_1._092 	:= PTB[220].IN_ConfigPresent;
//Recovery pump speed
HMI_CFG_PAM_1._116 := PPB[209].IN_ConfigPresent;
HMI_CFG_PAM_1._117 := PPB[209].IN_ConfigPresent;
HMI_CFG_PAM_1._118 := PPB[209].IN_ConfigPresent;

HMI_CFG_PAR_1._167	:= TRUE;
HMI_CFG_PAR_1._168	:= TRUE;
HMI_CFG_PAR_1._169	:= TRUE;
HMI_CFG_PAR_1._170	:= TRUE;
HMI_CFG_PAR_1._171	:= CFG_Par.Rinser.PressureNozzleControlInsertion OR CFG_Par.Rinser.PressureNozzleControlContinous;

//HMI Buttons//V4.A.A.1.7.0
HMI_RNS_SS2P[SS2P_SelAutoMan].Visibility		:= TRUE;
HMI_RNS_SS2P[SS2P_SelProduction].Visibility		:= TRUE;
HMI_RNS_SS2P[SS2P_SelDrain].Visibility			:= TRUE;
HMI_RNS_SS2P[SS2P_SelCIP].Visibility			:= FALSE; //CFG_Par.Rinser.CipPresent;
HMI_RNS_SS2P[SS2P_RNS_InsControl].Visibility	:= CFG_Par.Rinser.PressureNozzleControlInsertion;
HMI_RNS_SS2P[SS2P_RNS_ContControl].Visibility	:= CFG_Par.Rinser.PressureNozzleControlContinous;
HMI_RNS_PB[PB_CmdStart].Visibility				:= TRUE;
HMI_RNS_PB[PB_CmdStop].Visibility				:= TRUE;

(*RNS Nozzles Data Scroll //V4.A.A.1.7.0*)
VAR_RNS_MinPageData := 0;
VAR_RNS_MaxPageData := (HMI_PAC_1._200 / 15) -1;

HMI_RNS_PB[PB_RNS_PageDown].Visibility 	:= TRUE;
HMI_RNS_PB[PB_RNS_PageUp].Visibility 	:= TRUE;

VAR_RNS_NozzleInLastPage := (HMI_PAC_1._200 MOD 15);

IF VAR_RNS_NozzleInLastPage > 0 THEN
	VAR_RNS_MaxPageData := VAR_RNS_MaxPageData + 1;
END_IF
END_ACTION
TRANSITION FROM RNS_Cfg TO (RNSVar,Instruments,ModeSelection,MainSequencer,Valves,Pumps,DataTo):=
TRUE
END_TRANSITION
STEP RNSVar:
VAR_RNS_Blink1HzEp 		:= EDGEPOS(AID.DataOut.Blink1Hz);
VAR_RNS_PBResetEp		:= EDGEPOS(AID.DataOut.Reset);
END_STEP
STEP Instruments:
RNS_InstrFlow;
RNS_InstrPress;
RNS_InstrSaf;
RNS_InstrLevel; //v1.4
END_STEP
STEP ModeSelection:
RNS_ModeSelection;
END_STEP
STEP MainSequencer:
RNS_StepManager;
RNS_StepMove;
RNS_StepConfig;
RNS_StepStatus;
END_STEP
STEP Valves:
RNS_ValvesLogic;
RNS_ValvesFB;
RNS_ModulatingValvesPID;
END_STEP
STEP Pumps:
RNS_PumpsLogic;
RNS_PumpsPID;
RNS_PumpsFB;
END_STEP
STEP DataTo:
RNS_Alarm;
RNS_HMI;
RNS_DataOut;//V4.A.A.1.7.0
END_STEP
TRANSITION FROM (RNSVar,Instruments,ModeSelection,MainSequencer,Valves,Pumps,DataTo) TO RNS_Off:=
FALSE
END_TRANSITION
STEP RNS_Off:
ST_tmp_suspend(0);
END_STEP
TRANSITION FROM RNS_Off TO Step1:=
FALSE
END_TRANSITION
(* @SFCISJUMP := 'Step1' *)
END_PROGRAM
```

#### Devices.var
```iecst
(*VALVES*)
VAR
	AVB : ARRAY[MIN_CFG_AVx..MAX_CFG_AVx] OF Valve_Dig;
END_VAR
(*INSTRUMENTS - DIGITAL*)
VAR
	FSB : ARRAY[MIN_CFG_FSx..MAX_CFG_FSx] OF Digital_Obj;
	LSB : ARRAY[MIN_CFG_LSx..MAX_CFG_LSx] OF Digital_Obj;
END_VAR
(*RINSER RELEASED CLAMPS SAFETY*)
VAR
	_202DSB : Digital_Obj;
END_VAR
(*INSTRUMENTS - ANALOGIC*)
VAR
	PTB : ARRAY[MIN_CFG_PTx..MAX_CFG_PTx] OF Analog_In;
	LTB : ARRAY[MIN_CFG_LTx..MAX_CFG_LTx] OF Analog_In; (*vRMA*)
	FTB : ARRAY[MIN_CFG_FTx..MAX_CFG_FTx] OF Analog_In;
END_VAR
(*MOTORS*)
VAR
	PPB : ARRAY[MIN_CFG_VFD_PPx..MAX_CFG_VFD_PPx] OF Motor_FC280_Vfd;
	FB_PID_PPB209 : PID_Cont;
END_VAR
```

#### Types.typ - Local data types
```iecst
TYPE
	SEQ_Type : 	STRUCT
		Step : ARRAY[0..MAX_STEP_CFG]OF SEQ_Step_Type;
		ModeActual : UINT;
		StepActual : UINT;
		TON_Time_END : BOOL;
		T_Time_END : BOOL;
		TO_Time_END : BOOL;
		Laps_Done : BOOL;
		Cycles_Done : BOOL; (*All Cycles Done*)
	END_STRUCT;
	SEQ_Step_Type : 	STRUCT  (*V4.A.A.1.7.0*)
		Jump : ARRAY[0..MAX_JUMP_CFG]OF SEQ_Jump_Type;
		Config : SEQ_StepConfig_Type;
	END_STRUCT;
	SEQ_Jump_Type : 	STRUCT  (*V4.A.A.1.7.0*)
		Condition : BOOL;
		Number : UINT;
	END_STRUCT;
	VAR_RNS_SeqActualStep_Type :
		( (*V4.A.A.1.7.0*)
		RNS_SeqWait := 0,
		RNS_SeqPrdPriming := 5,
		RNS_SeqPrdPrimingTimeOut := 6,
		RNS_SeqSystemWaitCon := 7,
		RNS_SeqSystemOnTreatment := 11,
		RNS_SeqSystemTreatmentAlr := 26,
		RNS_SeqDrain := 22,
		RNS_SeqDrainDone := 23,
		RNS_SeqCip := 24, (*v1.4*)
		RNS_SeqCop := 25, (*v1.4*)
		RNS_SeqCipStopped := 30, (*v1.4*)
		RNS_SeqControl := 70, (*V4.A.A.1.7.0*)
		RNS_SeqBypass := 90, (*V4.A.A.1.7.0*)
		RNS_SeqStopped := 40
		);
END_TYPE

(*DEVICES*)

TYPE
	SEQ_Module_Type : 	STRUCT
		Device : SEQ_Device_Type;
		Mem : SEQ_Mem_Type;
		ITC : SEQ_ITC_Type;
	END_STRUCT;
	SEQ_Mem_Type : 	STRUCT
		ContainersStop : BOOL; (*Containers Stop Control (1 = Stop)*)
		ByPassRequest : BOOL; (*Rincer ByPass Request*)
		ByPassed : BOOL; (*Rincer ByPassed*)
		WaterTreatmentControl : BOOL; (*Water Spray Continous Mode*)
		AirTreatmentControl : BOOL; (*Air Spray Control Mode*)
		ControlInsercion : BOOL; (*Spray Control Insercion Mode*)
		ControlContinous : BOOL; (*Spray Control Continous Mode*)
		InsercionDevice : BOOL; (*Spray Control Device insercion Request*)
		SpeedReductionControl : BOOL; (*Spray Control Device insercion Request*)
		CopAfterCipRequest : BOOL; (*Cop Request After CIP*)
		PBAbortEnable : BOOL; (*PB Abort Sequence Enable*)
		PBStopEnable : BOOL; (*PB Stop Sequence Enable*)
		PBStartEnable : BOOL; (*PB Start Sequence Enable*)
		NoBoNoSprayInsercion : BOOL; (*No Bottle No Spray Insercion Device for Priming Nozle Rma tes*)
	END_STRUCT;
	SEQ_Device_Type : 	STRUCT
		AVB224 : Valve_Cmd_Type;
		AVB228 : Valve_Cmd_Type; (*V4.A.A.1.7.0*)
		AVB234 : Valve_Cmd_Type; (*vrma*)
		AVB261 : Valve_Cmd_Type;
		AVB264 : Valve_Cmd_Type; (*V4.A.A.1.7.0*)
		AVB265 : Valve_Cmd_Type; (*V4.A.A.1.7.0*)
		AVB266 : Valve_Cmd_Type; (*V4.A.A.1.7.0*)
		AVB267 : Valve_Cmd_Type; (*v1.4*)
		AVB268 : Valve_Cmd_Type; (*v1.4*)
		AVB273 : Valve_Cmd_Type; (*V4.A.A.1.7.0*)
		AVB294 : Valve_Cmd_Type;
		PPB209 : Seq_Motor_Type; (*v1.4*)
		RVB202_PID : PID_Type; (*V4.A.A.1.7.0*)
		PPB209_PID : PID_Type; (*v1.4*)
		LSB209 : Digital_In_Type; (*v1.4*)
		LSB210 : Digital_In_Type; (*v1.4*)
		LSB299 : Digital_In_Type; (*v1.4*)
		LTB202 : Analog_In_Type; (*vrma*)
		FSB201 : Digital_In_Type;
		FSB220 : Digital_In_Type;
		FTB201 : Analog_In_Type; (*v1.4*)
		FTB202 : Analog_In_Type; (*V4.A.A.1.7.0*)
		PTB220 : Analog_In_Type; (*V4.A.A.1.7.0*)
		PTB270 : Analog_In_Type; (*V4.A.A.1.7.0*)
		PTB290 : Analog_In_Type;
	END_STRUCT;
	SEQ_ITC_Type : 	STRUCT
		WTT_ProductRequest : BOOL; (*Production Mode Active*)
		WTT_ProductionRunning : BOOL; (*Filler Inlet Open - Start/Stop Overpressure Pump*)
	END_STRUCT;
	Analog_In_Type : 	STRUCT
		ALR_HighLimitEn : BOOL;
		ALR_HighLimitSP : REAL;
		ALR_LowLimitEn : BOOL;
		ALR_LowLimitSP : REAL;
		SP : REAL;
		CMP : USINT;
		MinDev : REAL;
		MaxDev : REAL;
	END_STRUCT;
	Digital_In_Type : 	STRUCT
		ALR : BOOL;
		WAIT_ON : BOOL;
		WAIT_OFF : BOOL;
	END_STRUCT;
	PID_Type : 	STRUCT
		PID_Enable : BOOL; (*PID Enable Condition*)
		PID_Mode : BOOL; (*PID Mode (1 = Auto - 0 = Manual)*)
		Auto_SP_Value : REAL;
		Auto_SP_MinDev : REAL;
		Auto_SP_MaxDev : REAL;
		FIX_Value : REAL;
	END_STRUCT;
	Seq_Motor_Type : 	STRUCT
		IN_Auto : BOOL; (*PID Enable Condition*)
		IN_AutoSP : REAL;
		IN_FixOut : BOOL;
		IN_FixOutValue : REAL;
	END_STRUCT;
	Valve_Cmd_Type : 	STRUCT
		AutoCnd : BOOL;
		EnableCnd : BOOL;
	END_STRUCT;
	Motor_Cmd_Type : 	STRUCT
		AutoCnd : BOOL;
	END_STRUCT;
END_TYPE
```

#### Variables.var - Local variables
```iecst
VAR
	TOF_StatusMachineRunning : TOF;
END_VAR
(*SELECTIONS*)
VAR
	VAR_RNS_FMDProduction : BOOL;
	VAR_RNS_FMDDrain : BOOL;
	VAR_RNS_FMDCip : BOOL;
	VAR_RNS_FMDCop : BOOL;
	VAR_RNS_FMDControl : BOOL; (*v4.A.A.A.1.6.15*)
	VAR_RNS_FMDByPass : BOOL; (*v4.A.A.A.1.6.15*)
	VAR_RNS_MemPBStart : BOOL;
	VAR_RNS_MemPBStop : BOOL;
	VAR_RNS_MemPBAbort : BOOL;
	VAR_RNS_MemPBSkipForward : BOOL;
	VAR_RNS_MemSSPause : BOOL;
END_VAR
(*AUXILIARY VARIABLES*)
VAR
	VAR_RNS_Blink1HzEp : BOOL;
	VAR_RNS_PBResetEp : BOOL;
	VAR_RNS_PBSelectionEnable : BOOL;
	VAR_RNS_TankLevelMedium : BOOL; (*v1.4*)
	VAR_RNS_TankLevelTooLow : BOOL;
	VAR_RNS_TankLevelLow : BOOL;
	VAR_RNS_TankLevelHigh : BOOL;
	VAR_RNS_InletOpen : BOOL;
	VAR_RNS_InletProductIncoming : BOOL;
	VAR_RNS_InletOpenCip : BOOL; (*v4.A.A.A.1.6.15*)
	VAR_RNS_OutletOpen : BOOL;
	VAR_RNS_ProductInletSafety : BOOL;
	VAR_RNS_ProductInletSafetyDelay : BOOL;
	VAR_RNS_ForIndex : UINT;
	VAR_RNS_MinPageData : INT; (*v4.A.A.A.1.6.15*)
	VAR_RNS_MaxPageData : INT; (*v4.A.A.A.1.6.15*)
	VAR_RNS_ActPageData : INT; (*v4.A.A.A.1.6.15*)
	VAR_RNS_NozzleInLastPage : INT; (*v4.A.A.A.1.6.15*)
	VAR_RNS_IndexVis : INT; (*v4.A.A.A.1.6.15*)
	VAR_RNS_IndexAlarm : INT; (*v4.A.A.A.1.6.15*)
	VAR_RNS_ContinousAirAlarm : UINT; (*v4.A.A.A.1.6.15*)
	VAR_RNS_ContinousWaterAlarm : UINT; (*v4.A.A.A.1.6.15*)
	VAR_RNS_InsercionAirAlarm : UINT; (*v4.A.A.A.1.6.15*)
	VAR_RNS_InsercionWaterAlarm : UINT; (*v4.A.A.A.1.6.15*)
	VAR_RNS_IndexReset : INT; (*v4.A.A.A.1.6.15*)
	VAR_RNS_TotalContainerEntered : UDINT; (*v4.A.A.A.1.6.15*)
	VAR_RNS_ControlRemainder_Cont : UDINT; (*v4.A.A.A.1.6.15*)
	VAR_RNS_ControlRemainder : UDINT; (*v4.A.A.A.1.6.15*)
	VAR_RNS_AirTreatment : BOOL; (*v4.A.A.A.1.6.15*)
	VAR_RNS_WaterTreatment : BOOL; (*v4.A.A.A.1.6.15*)
	VAR_RNS_CleaningActive : BOOL; (*v4.A.A.A.1.6.15*)
	VAR_RNS_ControlModeRequest : BOOL; (*v4.A.A.A.1.6.15*)
	VAR_RNS_ControlInsercionRequest : BOOL; (*v4.A.A.A.1.6.15*)
	VAR_RNS_ControlContinousRequest : BOOL; (*v4.A.A.A.1.6.15*)
	VAR_RNS_BypassRequest : BOOL; (*v4.A.A.A.1.6.15*)
	VAR_RNS_BypassCommand : BOOL; (*v4.A.A.A.1.6.15*)
	VAR_RNS_MemDisableAxisReq : BOOL; (*//RnsDisable*)
END_VAR
(*ALARM VARIABLES*)
VAR
	VAR_RNS_AirFlowTooHigh : BOOL; (*v4.A.A.A.1.6.15*)
	VAR_RNS_AirFlowTooLow : BOOL; (*v4.A.A.A.1.6.15*)
	VAR_RNS_AirFlowLowWarning : BOOL; (*v4.A.A.A.1.6.15*)
	VAR_RNS_WaterFlowTooHigh : BOOL;
	VAR_RNS_WaterFlowTooLow : BOOL;
	VAR_RNS_WaterFlowLowWarning : BOOL; (*v4.A.A.A.1.6.15*)
	VAR_RNS_WaterFlowMissing : BOOL; (*v4.A.A.A.1.6.15*)
	VAR_RNS_BottlesNotRinse : BOOL;
	VAR_RNS_AVB_ValveFault : BOOL;
END_VAR
(*AUXILIARY TIMERS*)
VAR
	TMR_TON_TankLowLevelLost : TON;
	TMR_TON_InletSafetyDelay : TON;
	TMR_TON_AirFlowLowLimitDelay : TON; (*v4.A.A.A.1.6.15*)
	TMR_TON_WtrFlowLowLimitDelay : TON; (*v4.A.A.A.1.6.15*)
	TMR_TON_WtrFlowSwitchDelay : TON; (*v4.A.A.A.1.6.15*)
	TMR_TON_FlipWait : TON;
	TMR_TOF_FlipWork : TOF;
END_VAR
(*PID*)
VAR CONSTANT
	PID_MODE_CIP : USINT := 0;
	PID_MODE_PRD : USINT := 1;
END_VAR
VAR
	FB_PID_RVB202 : ARRAY[0..3] OF PID_Cont; (*v4.A.A.A.1.6.15*)
	FB_PID_PPB220 : ARRAY[0..3] OF PID_Cont;
END_VAR
(*SAFETY STATUS*)
VAR
	VAR_RNS_ValveEnable : BOOL;
	VAR_RNS_ValveEnableCip : BOOL; (*v4.A.A.A.1.6.15*)
	VAR_RNS_PumpEnable : BOOL;
	VAR_RNS_MotorEnable : BOOL;
	VAR_SetReset : SR; (*v1.4*)
	VAR_RNS_RVB202Auto : BOOL; (*v4.A.A.A.1.6.15*)
END_VAR
```

#### VariablesSeq.var - Local variables
```iecst
(*SEQUENCER*)
VAR
	FB_RNS_SEQ : Sequencer_v2;
	VAR_RNS_SEQ_Step : SEQ_Type;
	VAR_RNS_SEQ : SEQ_Module_Type;
	VAR_RNS_SeqProdStopAlarm : BOOL;
	VAR_RNS_SeqProdStopRequest : BOOL;
	VAR_RNS_SeqProdAbortRequest : BOOL;
	VAR_RNS_SeqCipStopAlarm : BOOL;
	VAR_RNS_SeqCipStopRequest : BOOL;
	VAR_RNS_SeqCipAbortRequest : BOOL;
	VAR_RNS_SeqDrainStopAlarm : BOOL;
	VAR_RNS_SeqDrainStopRequest : BOOL;
	VAR_RNS_SeqDrainAbortRequest : BOOL;
	VAR_RNS_SeqControlStopAlarm : BOOL; (*v4.A.A.A.1.6.15*)
	VAR_RNS_SeqControlStopRequest : BOOL; (*v4.A.A.A.1.6.15*)
	VAR_RNS_SeqControlAbortRequest : BOOL; (*v4.A.A.A.1.6.15*)
	VAR_RNS_SeqBypassStopAlarm : BOOL; (*v4.A.A.A.1.6.15*)
	VAR_RNS_SeqBypassAbortRequest : BOOL; (*v4.A.A.A.1.6.15*)
	VAR_index : UINT;
	VAR_RNS_SeqActualStep : UINT;(*v4.A.A.A.1.6.15*)
	VAR_RNS_SeqCyclesCounter : UDINT;
END_VAR
(*MODE VARIABLES*)
VAR
	VAR_RNS_ModeWait : BOOL;
	VAR_RNS_ModeProduction : BOOL;
	VAR_RNS_ModeCip : BOOL;
	VAR_RNS_ModeRinse : BOOL;
	VAR_RNS_ModeDrain : BOOL;
	VAR_RNS_ModeCop : BOOL;
	VAR_RNS_ModeControl : BOOL;(*v4.A.A.A.1.6.15*)
	VAR_RNS_ModeBypass : BOOL; (*v4.A.A.A.1.6.15*)
	VAR_RNS_MemProdDrain : BOOL;
	VAR_RNS_MemProdControl : BOOL;
	VAR_RNS_MemRinserByPassed : BOOL;(*v4.A.A.A.1.6.15*)
	VAR_RNS_MemRinserInserted : BOOL; (*v4.A.A.A.1.6.15*)
	VAR_RNS_ModeFiltersSterilization : BOOL;
	VAR_RNS_ModeDeEnergization : BOOL;
	VAR_RNS_ModeWaitOperator : BOOL;
END_VAR
(*STEP VARIABLES*)
(*Production*)
VAR
	VAR_RNS_StepProdStartUp : BOOL;
	VAR_RNS_StepProdStartUpLampCtrl : BOOL;
	VAR_RNS_StepProdStartUpLampFault : BOOL;
	VAR_RNS_StepProdProducing : BOOL;
	VAR_RNS_StepProdSprayRequest : BOOL;
	VAR_RNS_StepProdLampOnDischarge : BOOL;
	VAR_RNS_StepProdStopped : BOOL;
	VAR_RNS_StepProdAborted : BOOL;
END_VAR
(*Cip*)
VAR
	VAR_RNS_StepCipFilling : BOOL;
	VAR_RNS_StepCipCleaning : BOOL;
	VAR_RNS_StepCipDraining : BOOL;
	VAR_RNS_StepCipRecovery : BOOL;
	VAR_RNS_StepCipPipeFlooding : BOOL;
	VAR_RNS_StepCipPipeDischarge : BOOL;
	VAR_RNS_StepCipFlooding : BOOL;
	VAR_RNS_StepCipFlooded : BOOL;
	VAR_RNS_StepCipStopped : BOOL;
	VAR_RNS_StepCipAborted : BOOL;
	VAR_RNS_StepCipEnded : BOOL;
END_VAR
(*Drain*)
VAR
	VAR_RNS_StepDrainStopped : BOOL;
	VAR_RNS_StepDrainAborted : BOOL;
END_VAR
(*Control*)
VAR
	VAR_RNS_StepControl : BOOL;(*v4.A.A.A.1.6.15*)
	VAR_RNS_StepControlDone : BOOL;(*v4.A.A.A.1.6.15*)
	VAR_RNS_StepCtrlCipDone : BOOL; (*v4.A.A.A.1.6.15*)
	VAR_RNS_StepControlStopped : BOOL;(*v4.A.A.A.1.6.15*)
	VAR_RNS_StepControlAborted : BOOL;(*v4.A.A.A.1.6.15*)
END_VAR
(*By Pass*)
VAR
	VAR_RNS_StepByPassed : BOOL;(*v4.A.A.A.1.6.15*)
	VAR_RNS_StepBypassAborted : BOOL;(*v4.A.A.A.1.6.15*)
END_VAR
(*Motion*)
VAR
	VAR_RNS_StepMotorization : BOOL; (*//RnsDisable*)
END_VAR
```

#### RNS_InstrFlow.st
```iecst
ACTION RNS_InstrFlow:
//FSB201 RINSER
	FSB[201](
	IN_ConfigPresent 	:= FSB[201].IN_ConfigPresent,
	IN_Alarm 			:= TNK.DataOut.ProdMode AND MNM.DataOut.MachineRunning AND AVB[228].IN_AutoCnd,
	IN_AlarmOnReq		:= FALSE,
	IN_AlarmOffReq 		:= (AVB[228].IN_ConfigPresent AND TNK.DataOut.ProdMode AND MNM.DataOut.MachineRunning AND AVB[228].IN_AutoCnd),
	IN_SwitchDelay 		:= T#50ms,
	IN_WaitOn 			:= AVB[228].IN_AutoCnd,
	IN_WaitOff 			:= FALSE,
	IN_Reset	 		:= VAR_RNS_PBResetEp,
	IN_MaskEn 			:= TRUE,
	IO 					:= IO_FSB[201],
	HMI 				:= HMI_FSB[201]
	);

//FSB220 RINSER SPRAY FLOWSWITCH

	//Alarm Delay//V4.A.A.1.7.0
	TMR_TON_WtrFlowSwitchDelay.IN := VAR_RNS_SEQ.Device.FSB220.ALR  AND SFT.DataOut.NoBottleNoSprayActive AND VAR_RNS_InletProductIncoming;//vrma
	TMR_TON_WtrFlowSwitchDelay.PT := T#5s;
	TMR_TON_WtrFlowSwitchDelay();

	FSB[220](//V4.A.A.1.7.0
	IN_ConfigPresent 	:= FSB[220].IN_ConfigPresent,
	IN_Alarm 			:= TMR_TON_WtrFlowSwitchDelay.Q,
	IN_AlarmOnReq		:= FALSE,
	IN_AlarmOffReq 		:= TMR_TON_WtrFlowSwitchDelay.Q,
	IN_SwitchDelay 		:= T#50ms,
	IN_WaitOn 			:= VAR_RNS_SEQ.Device.FSB220.WAIT_ON,
	IN_WaitOff 			:= FALSE,
	IN_Reset	 		:= VAR_RNS_PBResetEp,
	IN_MaskEn 			:= TRUE,
	IO 					:= IO_FSB[220],
	HMI 				:= HMI_FSB[220]
	);

	IF FSB[220].OUT_Alarm THEN//V4.A.A.1.7.0
		VAR_RNS_WaterFlowMissing :=  TRUE ;
	ELSIF VAR_RNS_PBResetEp THEN
		VAR_RNS_WaterFlowMissing :=  FALSE;
	END_IF

//FTB201 RINSER FLOW TRASMITTER AIR

	//Alarm Delay
	TMR_TON_AirFlowLowLimitDelay.IN := VAR_RNS_SEQ.Device.FTB201.ALR_LowLimitEn;
	TMR_TON_AirFlowLowLimitDelay.PT := T#5s;
	TMR_TON_AirFlowLowLimitDelay();

	IF TMR_TON_AirFlowLowLimitDelay.Q THEN
		FTB[201].IN_LowLimitDelay := T#1s;
	ELSE
		FTB[201].IN_LowLimitDelay := T#5s;
	END_IF

	FTB[201](
	IN_ConfigPresent 	:= FTB[201].IN_ConfigPresent,
	IN_EngScale 		:= FTB[201].IN_EngScale,
	IN_CompareMode 		:= VAR_RNS_SEQ.Device.FTB201.CMP,
	IN_AlarmEn 			:= TRUE,
	IN_MaskEn 			:= TRUE,
	IN_Reset 			:= VAR_RNS_PBResetEp,
	IN_ActualSP 		:= VAR_RNS_SEQ.Device.FTB201.SP,
	IN_MinDev 			:= VAR_RNS_SEQ.Device.FTB201.MinDev,
	IN_MaxDev 			:= VAR_RNS_SEQ.Device.FTB201.MaxDev,
	IN_WaitDelay 		:= T#500ms,
	IN_HighLimitEn 		:= VAR_RNS_SEQ.Device.FTB201.ALR_HighLimitEn,
	IN_HighLimitSP 		:= VAR_RNS_SEQ.Device.FTB201.ALR_HighLimitSP,
	IN_HighLimitHyst 	:= 0.0,
	IN_HighLimitDelay 	:= T#1s,
	IN_LowLimitEn 		:= VAR_RNS_SEQ.Device.FTB201.ALR_LowLimitEn,
	IN_LowLimitSP 		:= VAR_RNS_SEQ.Device.FTB201.ALR_LowLimitSP,
	IN_LowLimitHyst 	:= 0.0,
	IN_LowLimitDelay 	:= FTB[201].IN_LowLimitDelay,
	IN_TotPulseWeight 	:= 0.0,
	IN_TotType 			:= 0,
	IN_PLCCounterEn 	:= FALSE,
	IN_PLCCounterSP 	:= 0.0,
	IN_PLCCounterReset	:= FALSE,
	IN_HMITotEn 		:= FALSE,
	IN_HMITotReset 		:= FALSE,
	IO 					:= IO_FTB[201],
	HMI 				:= HMI_FTB[201]
	);

	VAR_RNS_AirFlowTooHigh := FTB[201].OUT_HighLimit;

	IF FTB[201].OUT_LowLimit THEN
		VAR_RNS_AirFlowTooLow	:= TRUE;
	ELSIF VAR_RNS_PBResetEp THEN
		VAR_RNS_AirFlowTooLow	:= FALSE;
	END_IF

	VAR_RNS_AirFlowLowWarning := NOT FTB[201].OUT_SpReached AND (FTB[201].OUT_ActValue < FTB[201].IN_ActualSP);

//FTB202 RINSER FLOW TRASMITTER H2O

	//Alarm Delay
	TMR_TON_WtrFlowLowLimitDelay.IN := VAR_RNS_SEQ.Device.FTB202.ALR_LowLimitEn AND SFT.DataOut.NoBottleNoSprayActive AND VAR_RNS_InletProductIncoming;//vrma
	TMR_TON_WtrFlowLowLimitDelay.PT := T#5s;
	TMR_TON_WtrFlowLowLimitDelay();

	IF TMR_TON_WtrFlowLowLimitDelay.Q THEN
		FTB[202].IN_LowLimitDelay := T#1s;
	ELSE
		FTB[202].IN_LowLimitDelay := T#5s;
	END_IF

	FTB[202](
	IN_ConfigPresent 	:= FTB[202].IN_ConfigPresent,
	IN_EngScale 		:= FTB[202].IN_EngScale,
	IN_CompareMode 		:= VAR_RNS_SEQ.Device.FTB202.CMP,
	IN_AlarmEn 			:= TRUE,
	IN_MaskEn 			:= TRUE,
	IN_Reset 			:= VAR_RNS_PBResetEp,
	IN_ActualSP 		:= VAR_RNS_SEQ.Device.FTB202.SP,
	IN_MinDev 			:= VAR_RNS_SEQ.Device.FTB202.MinDev,
	IN_MaxDev 			:= VAR_RNS_SEQ.Device.FTB202.MaxDev,
	IN_WaitDelay 		:= T#500ms,
	IN_HighLimitEn 		:= VAR_RNS_SEQ.Device.FTB202.ALR_HighLimitEn AND SFT.DataOut.NoBottleNoSprayActive,
	IN_HighLimitSP 		:= VAR_RNS_SEQ.Device.FTB202.ALR_HighLimitSP,
	IN_HighLimitHyst 	:= 0.0,
	IN_HighLimitDelay 	:= T#1s,
	IN_LowLimitEn 		:= VAR_RNS_SEQ.Device.FTB202.ALR_LowLimitEn AND SFT.DataOut.NoBottleNoSprayActive AND VAR_RNS_InletProductIncoming,
	IN_LowLimitSP 		:= VAR_RNS_SEQ.Device.FTB202.ALR_LowLimitSP,
	IN_LowLimitHyst 	:= 0.0,
	IN_LowLimitDelay 	:= FTB[202].IN_LowLimitDelay,
	IN_TotPulseWeight 	:= 0.0,
	IN_TotType 			:= 0,
	IN_PLCCounterEn 	:= FALSE,
	IN_PLCCounterSP 	:= 0.0,
	IN_PLCCounterReset	:= FALSE,
	IN_HMITotEn 		:= FALSE,
	IN_HMITotReset 		:= FALSE,
	IO 					:= IO_FTB[202],
	HMI 				:= HMI_FTB[202]
	);

	VAR_RNS_WaterFlowTooHigh := FTB[202].OUT_HighLimit;

	IF FTB[202].OUT_LowLimit THEN
		VAR_RNS_WaterFlowTooLow	:= NOT SFT.DataOut.MachineEmpty;
	ELSIF VAR_RNS_PBResetEp THEN
		VAR_RNS_WaterFlowTooLow	:= FALSE;
	END_IF

	IF VAR_RNS_SEQ.Device.FTB202.ALR_LowLimitEn AND SFT.DataOut.NoBottleNoSprayActive AND VAR_RNS_InletProductIncoming  THEN//vrma
		VAR_RNS_WaterFlowLowWarning := NOT FTB[202].OUT_SpReached AND (FTB[202].OUT_ActValue < FTB[202].IN_ActualSP);
	ELSE
		VAR_RNS_WaterFlowLowWarning := FALSE;
	END_IF

END_ACTION
```

#### RNS_InstrPress.st
```iecst
ACTION RNS_InstrPress:
	//H2O
	PTB[220](
	IN_ConfigPresent 	:= PTB[220].IN_ConfigPresent,
	IN_EngScale 		:= PTB[220].IN_EngScale,
	IN_CompareMode 		:= VAR_RNS_SEQ.Device.PTB220.CMP,
	IN_AlarmEn 			:= TRUE,
	IN_MaskEn 			:= TRUE,
	IN_Reset 			:= VAR_RNS_PBResetEp,
	IN_ActualSP 		:= VAR_RNS_SEQ.Device.PTB220.SP,
	IN_MinDev 			:= VAR_RNS_SEQ.Device.PTB220.MinDev,
	IN_MaxDev 			:= VAR_RNS_SEQ.Device.PTB220.MaxDev,
	IN_WaitDelay 		:= T#500ms,
	IN_HighLimitEn 		:= VAR_RNS_SEQ.Device.PTB220.ALR_HighLimitEn,
	IN_HighLimitSP 		:= VAR_RNS_SEQ.Device.PTB220.ALR_HighLimitSP,
	IN_HighLimitHyst 	:= 0.0,
	IN_HighLimitDelay 	:= T#1s,
	IN_LowLimitEn 		:= VAR_RNS_SEQ.Device.PTB220.ALR_LowLimitEn,
	IN_LowLimitSP 		:= VAR_RNS_SEQ.Device.PTB220.ALR_LowLimitSP,
	IN_LowLimitHyst 	:= 0.0,
	IN_LowLimitDelay 	:= T#1s,
	IN_TotPulseWeight 	:= 0.0,
	IN_TotType 			:= 0,
	IN_PLCCounterEn 	:= FALSE,
	IN_PLCCounterSP 	:= 0.0,
	IN_PLCCounterReset	:= FALSE,
	IN_HMITotEn 		:= FALSE,
	IN_HMITotReset 		:= FALSE,
	IO 					:= IO_PTB[220],
	HMI 				:= HMI_PTB[220]
	);

	//Air//V4.A.A.1.7.0
	PTB[270](
	IN_ConfigPresent 	:= PTB[270].IN_ConfigPresent,
	IN_EngScale 		:= PTB[270].IN_EngScale,
	IN_CompareMode 		:= VAR_RNS_SEQ.Device.PTB270.CMP,
	IN_AlarmEn 			:= TRUE,
	IN_MaskEn 			:= TRUE,
	IN_Reset 			:= VAR_RNS_PBResetEp,
	IN_ActualSP 		:= VAR_RNS_SEQ.Device.PTB270.SP,
	IN_MinDev 			:= VAR_RNS_SEQ.Device.PTB270.MinDev,
	IN_MaxDev 			:= VAR_RNS_SEQ.Device.PTB270.MaxDev,
	IN_WaitDelay 		:= T#500ms,
	IN_HighLimitEn 		:= VAR_RNS_SEQ.Device.PTB270.ALR_HighLimitEn,
	IN_HighLimitSP 		:= VAR_RNS_SEQ.Device.PTB270.ALR_HighLimitSP,
	IN_HighLimitHyst 	:= 0.0,
	IN_HighLimitDelay 	:= T#1s,
	IN_LowLimitEn 		:= VAR_RNS_SEQ.Device.PTB270.ALR_LowLimitEn,
	IN_LowLimitSP 		:= VAR_RNS_SEQ.Device.PTB270.ALR_LowLimitSP,
	IN_LowLimitHyst 	:= 0.0,
	IN_LowLimitDelay 	:= T#1s,
	IN_TotPulseWeight 	:= 0.0,
	IN_TotType 			:= 0,
	IN_PLCCounterEn 	:= FALSE,
	IN_PLCCounterSP 	:= 0.0,
	IN_PLCCounterReset	:= FALSE,
	IN_HMITotEn 		:= FALSE,
	IN_HMITotReset 		:= FALSE,
	IO 					:= IO_PTB[270],
	HMI 				:= HMI_PTB[270]
	);

	//Check Pressure on Bottle Shower vrma
	PTB[290](
	IN_ConfigPresent 	:= PTB[290].IN_ConfigPresent,
	IN_EngScale 		:= PTB[290].IN_EngScale,
	IN_CompareMode 		:= 2,
	IN_AlarmEn 			:= TRUE,
	IN_MaskEn 			:= TRUE,
	IN_Reset 			:= VAR_RNS_PBResetEp,
	IN_ActualSP 		:= 2.5,
	IN_MinDev 			:= 0.3,
	IN_MaxDev 			:= 0.3,
	IN_WaitDelay 		:= T#500ms,
	IN_HighLimitEn 		:= FALSE,
	IN_HighLimitSP 		:= 0.0,
	IN_HighLimitHyst 	:= 0.0,
	IN_HighLimitDelay 	:= T#1s,
	IN_LowLimitEn 		:= TRUE,
	IN_LowLimitSP 		:= 2.0,
	IN_LowLimitHyst 	:= 0.0,
	IN_LowLimitDelay 	:= T#3s,
	IN_TotPulseWeight 	:= 0.0,
	IN_TotType 			:= 0,
	IN_PLCCounterEn 	:= FALSE,
	IN_PLCCounterSP 	:= 0.0,
	IN_PLCCounterReset	:= FALSE,
	IN_HMITotEn 		:= FALSE,
	IN_HMITotReset 		:= FALSE,
	IO 					:= IO_PTB[290],
	HMI 				:= HMI_PTB[290]
	);

END_ACTION
```

#### RNS_InstrSaf.st
```iecst
ACTION RNS_InstrSaf:
//Rinser Released Pairs Safety
	_202DSB(
	IN_ConfigPresent 	:= FSB[201].IN_ConfigPresent,
	IN_Alarm 			:= TRUE,
	IN_AlarmOnReq		:= FALSE,
	IN_AlarmOffReq 		:= TRUE,
	IN_SwitchDelay 		:= T#1ms,
	IN_WaitOn 			:= TRUE,
	IN_WaitOff 			:= FALSE,
	IN_Reset	 		:= VAR_RNS_PBResetEp,
	IN_MaskEn 			:= TRUE,
	IO 					:= IO_202DSB,
	HMI 				:= HMI_202DSB
	);
END_ACTION
```

#### RNS_InstrLevel.st
```iecst
ACTION RNS_InstrLevel:
//LSB209 COOLING RECOVERY TANK HIGH LEVEL PROBE
	LSB[209](
	IN_ConfigPresent 	:= LSB[209].IN_ConfigPresent,
	IN_Alarm 			:= VAR_RNS_SEQ.Device.LSB209.ALR,
	IN_AlarmOnReq		:= LSB[209].IN_WaitOff,
	IN_AlarmOffReq 		:= LSB[209].IN_WaitOn,
	IN_SwitchDelay 		:= T#500ms,
	IN_WaitOn 			:= VAR_RNS_SEQ.Device.LSB209.WAIT_ON,
	IN_WaitOff 			:= VAR_RNS_SEQ.Device.LSB209.WAIT_OFF,
	IN_OnDelay			:= T#5s,
	IN_OffDelay			:= T#5s,
	IN_Reset	 		:= VAR_RNS_PBResetEp,
	IN_MaskEn 			:= TRUE,
	IO 					:= IO_LSB[209],
	HMI 				:= HMI_LSB[209]
	);

//LSB210 RECOVERY TANK LOW LEVEL PROBE
	LSB[210](
	IN_ConfigPresent 	:= LSB[210].IN_ConfigPresent,
	IN_Alarm 			:= VAR_RNS_SEQ.Device.LSB210.ALR,
	IN_AlarmOnReq		:= LSB[210].IN_WaitOn,
	IN_AlarmOffReq 		:= LSB[210].IN_WaitOff,
	IN_SwitchDelay 		:= T#500ms,
	IN_WaitOn 			:= VAR_RNS_SEQ.Device.LSB210.WAIT_ON,
	IN_WaitOff 			:= VAR_RNS_SEQ.Device.LSB210.WAIT_OFF,
	IN_OnDelay			:= T#1s,
	IN_OffDelay			:= T#1s,
	IN_Reset	 		:= VAR_RNS_PBResetEp,
	IN_MaskEn 			:= TRUE,
	IO 					:= IO_LSB[210],
	HMI 				:= HMI_LSB[210]
	);

	TMR_TON_TankLowLevelLost(
	IN := LSB[210].OUT_OffDelayed OR LTB[202].OUT_ActValue < 3.0 ,
	PT := t#3s
	);

	VAR_RNS_TankLevelTooLow		:= TMR_TON_TankLowLevelLost.Q;
	VAR_RNS_TankLevelLow		:= LTB[202].OUT_ActValue > 30.0;
	VAR_RNS_TankLevelHigh		:= LSB[209].OUT_OnDelayed OR (LTB[202].OUT_ActValue > 70.0);
	VAR_RNS_TankLevelMedium		:= LSB[299].OUT_OnDelayed OR (LTB[202].OUT_ActValue > 50.0);

//LSB299 RECOVERY TANK MEDIUM LEVEL PROBE //v1.4
	LSB[299](
	IN_ConfigPresent 	:= LSB[299].IN_ConfigPresent,
	IN_Alarm 			:= VAR_RNS_SEQ.Device.LSB299.ALR,
	IN_AlarmOnReq		:= LSB[299].IN_WaitOn,
	IN_AlarmOffReq 		:= LSB[299].IN_WaitOff,
	IN_SwitchDelay 		:= T#500ms,
	IN_WaitOn 			:= VAR_RNS_SEQ.Device.LSB299.WAIT_ON,
	IN_WaitOff 			:= VAR_RNS_SEQ.Device.LSB299.WAIT_OFF,
	IN_Reset	 		:= VAR_RNS_PBResetEp,
	IN_MaskEn 			:= TRUE,
	IO 					:= IO_LSB[299],
	HMI 				:= HMI_LSB[299]
	);

	LTB[202](//vRMA
	IN_ConfigPresent 	:= LTB[202].IN_ConfigPresent,
	IN_FaultOutMode 	:= 0,
	IN_EngScale 		:= LTB[202].IN_EngScale,
	IN_AlarmEn 			:= TRUE,
	IN_MaskEn 			:= TRUE,
	IN_Reset 			:= VAR_RNS_PBResetEp,
	IN_HighLimitEn 		:= VAR_RNS_SEQ.Device.LTB202.ALR_HighLimitEn,
	IN_HighLimitSP 		:= VAR_RNS_SEQ.Device.LTB202.ALR_HighLimitSP,
	(*IN_HighLimitHyst 	:= VAR_RNS_SEQ.Device.LTB202.,*)
	IN_HighLimitDelay 	:= T#100ms,
	IN_LowLimitEn 		:= VAR_RNS_SEQ.Device.LTB202.ALR_LowLimitEn,
	IN_LowLimitSP 		:= VAR_RNS_SEQ.Device.LTB202.ALR_LowLimitSP,
	IN_LowLimitHyst 	:= 2.0,
	IN_LowLimitDelay 	:= T#100ms,
	IN_TotPulseWeight 	:= FALSE,
	IN_TotType 			:= 0,
	IN_PLCCounterEn 	:= FALSE,
	IN_PLCCounterSP 	:= 0.0,
	IN_PLCCounterReset	:= FALSE,
	IN_HMITotEn 		:= FALSE,
	IN_HMITotReset 		:= FALSE,
	IO 					:= IO_LTB[202],
	HMI 				:= HMI_LTB[202]
	);

END_ACTION
```

#### RNS_ModeSelection.st
```iecst
ACTION RNS_ModeSelection:
	IF NOT HMI_SS2P[SS2P_HMI_SelEnable].ON THEN
		HMI_RNS_SS2P[SS2P_SelAutoMan].ON := FALSE;
	END_IF

	//WAIT MODE
	IF EDGEPOS(VAR_RNS_SeqPermanent.SeqActualStep = 0) THEN
		FOR VAR_RNS_ForIndex:=1 TO 6 DO //ALL OTHER SELECTIONS RESET
			HMI_RNS_SS2P[VAR_RNS_ForIndex].ON := FALSE;
		END_FOR;
	END_IF

	//TREATMENT ACTIVE
	VAR_RNS_WaterTreatment := (HMI_RNS_SS2P[SS2P_SelAutoMan].ON AND (HMI_RNS_ManualSelection.Value < 2)) OR (NOT HMI_RNS_SS2P[SS2P_SelAutoMan].ON AND(HMI_PAR_1._170 < 2));
	//CONTROL TYPE REQUEST
	VAR_RNS_ControlInsercionRequest := (HMI_RNS_SS2P[SS2P_SelAutoMan].ON AND HMI_RNS_SS2P[SS2P_RNS_InsControl].ON) OR (NOT HMI_RNS_SS2P[SS2P_SelAutoMan].ON AND VAR_RNS_WaterTreatment);//HMI_PAR_1._171 > 0
	VAR_RNS_ControlContinousRequest	:= (HMI_RNS_SS2P[SS2P_SelAutoMan].ON AND HMI_RNS_SS2P[SS2P_RNS_ContControl].ON) OR (NOT HMI_RNS_SS2P[SS2P_SelAutoMan].ON AND VAR_RNS_AirTreatment);//HMI_PAR_1._171 < 1

	//On RMB220 Insercion control is for Water only and Continous control is for Air only
	IF HMI_RNS_SS2P[SS2P_SelAutoMan].ON THEN
		IF HMI_RNS_SS2P[SS2P_RNS_InsControl].ON THEN
			HMI_RNS_ManualSelection.Value := 1;//Water Only
		END_IF
		IF HMI_RNS_SS2P[SS2P_RNS_ContControl].ON THEN
			HMI_RNS_ManualSelection.Value := 2;//Air Only
		END_IF
	ELSE
		HMI_RNS_ManualSelection.Value := 0;
	END_IF

	//SS2P PRODUCTION MODE SELECTION
	VAR_RNS_FMDProduction := (HMI_RNS_SS2P[SS2P_SelProduction].ON AND HMI_RNS_SS2P[SS2P_SelAutoMan].ON) OR
								(TNK.DataOut.ProdMode AND NOT HMI_RNS_SS2P[SS2P_SelAutoMan].ON);//vrma

	IF EDGEPOS(VAR_RNS_FMDProduction) THEN //ALL OTHER SELECTIONS RESET
		FOR VAR_RNS_ForIndex:=1 TO 6 DO//V4.A.A.1.7.0
			IF VAR_RNS_ForIndex<>SS2P_SelProduction THEN
				HMI_RNS_SS2P[VAR_RNS_ForIndex].ON := FALSE;
			END_IF
		END_FOR;
	END_IF

	//SS2P CONTROL MODE SELECTION //V4.A.A.1.7.0
	VAR_RNS_TotalContainerEntered := HMI_CounterDataTotal.ContainersCounters.CounterData[ContainersEntered].CounterValue;
	VAR_RNS_ControlRemainder := (VAR_RNS_TotalContainerEntered MOD (REAL_TO_UDINT(HMI_PAM_1._090)) AND CFG_Par.Rinser.PressureNozzleControlInsertion);//vrma
	VAR_RNS_ControlRemainder_Cont := (VAR_RNS_TotalContainerEntered MOD (REAL_TO_UDINT(HMI_PAM_1._091))AND CFG_Par.Rinser.PressureNozzleControlContinous);//vrma
	IF 	NOT VAR_RNS_FMDControl AND
		((VAR_RNS_ControlRemainder = 0)  AND (HMI_PAM_1._090 <> 0) AND (VAR_RNS_TotalContainerEntered > REAL_TO_UDINT(HMI_PAM_1._090))) OR //CHECK FRA
		((VAR_RNS_ControlRemainder_Cont = 0) AND (HMI_PAM_1._091 <> 0) AND (VAR_RNS_TotalContainerEntered > REAL_TO_UDINT(HMI_PAM_1._091))) THEN //CHECK FRA
		VAR_RNS_ControlModeRequest := TRUE;
	END_IF

	IF VAR_RNS_StepControlDone THEN
		VAR_RNS_ControlModeRequest := FALSE;
	END_IF

	VAR_RNS_FMDControl := 	(HMI_RNS_SS2P[SS2P_SelAutoMan].ON AND (HMI_RNS_SS2P[SS2P_RNS_InsControl].ON OR HMI_RNS_SS2P[SS2P_RNS_ContControl].ON)) OR
							(TNK.DataOut.ProdMode AND NOT HMI_RNS_SS2P[SS2P_SelAutoMan].ON AND VAR_RNS_ControlModeRequest);//vrma

	IF EDGEPOS (VAR_RNS_FMDControl) THEN //ALL OTHER SELECTIONS RESET
		FOR VAR_RNS_ForIndex:=1 TO 6 DO
			IF HMI_RNS_SS2P[SS2P_RNS_InsControl].ON THEN
				IF VAR_RNS_ForIndex<>SS2P_RNS_InsControl THEN
					HMI_RNS_SS2P[VAR_RNS_ForIndex].ON := FALSE;
				END_IF
			ELSIF HMI_RNS_SS2P[SS2P_RNS_ContControl].ON THEN
				IF VAR_RNS_ForIndex<>SS2P_RNS_ContControl THEN
					HMI_RNS_SS2P[VAR_RNS_ForIndex].ON := FALSE;
				END_IF
			END_IF
		END_FOR;
	END_IF

	//SS2P DRAIN MODE SELECTION
	VAR_RNS_FMDDrain := (HMI_RNS_SS2P[SS2P_SelDrain].ON AND HMI_RNS_SS2P[SS2P_SelAutoMan].ON) OR
						(TNK.DataOut.DrainMode AND NOT HMI_RNS_SS2P[SS2P_SelAutoMan].ON);

	IF EDGEPOS(VAR_RNS_FMDDrain) THEN //ALL OTHER SELECTIONS RESET
		FOR VAR_RNS_ForIndex:=1 TO 6 DO
			IF VAR_RNS_ForIndex<>SS2P_SelDrain THEN
				HMI_RNS_SS2P[VAR_RNS_ForIndex].ON := FALSE;
			END_IF
		END_FOR;
	END_IF

	//SS2P CLEANING MODE SELECTION
	VAR_RNS_FMDCip := 	(HMI_RNS_SS2P[SS2P_SelCIP].ON AND HMI_RNS_SS2P[SS2P_SelAutoMan].ON) OR TNK.DataOut.CipMode; // leo  AND NOT TNK.DataOut.DisableCipRinser; //mixer

	VAR_RNS_CleaningActive := VAR_RNS_FMDCip AND (VAR_RNS_InletOpen);//vrma da controllare

	IF EDGEPOS(VAR_RNS_FMDCip) THEN //ALL OTHER SELECTIONS RESET
		FOR VAR_RNS_ForIndex:=1 TO 6 DO//V4.A.A.1.7.0
			IF VAR_RNS_ForIndex<>SS2P_SelCIP THEN
				HMI_RNS_SS2P[VAR_RNS_ForIndex].ON := FALSE;
			END_IF
		END_FOR;
	END_IF

	//PB START
	IF HMI_RNS_SS2P[SS2P_SelAutoMan].ON THEN
		VAR_RNS_MemPBStart := EDGEPOS(HMI_RNS_PB[PB_CmdStart].ON);
	ELSE
		VAR_RNS_MemPBStart := EDGEPOS(VAR_RNS_FMDProduction) OR EDGEPOS(VAR_RNS_FMDDrain) OR EDGEPOS(VAR_RNS_FMDCip);
	END_IF

	//PB STOP
	VAR_RNS_MemPBStop	:= EDGEPOS(HMI_RNS_PB[PB_CmdStop].ON);

	//PB ABORT
	VAR_RNS_MemPBAbort	:= EDGEPOS(HMI_RNS_PB[PB_CmdAbort].ON);

	//PB SKIP FORWARD
	VAR_RNS_MemPBSkipForward	:= EDGEPOS(HMI_RNS_PB[PB_CmdSkip].ON);

	//PB PAUSE
	IF EDGEPOS(HMI_RNS_PB[PB_CmdPause].ON) THEN
		IF VAR_RNS_MemSSPause THEN
			HMI_RNS_PB[PB_CmdPause].LampON	:= FALSE;
		ELSE
			HMI_RNS_PB[PB_CmdPause].LampON	:= TRUE;
		END_IF
	END_IF

	VAR_RNS_MemSSPause:= HMI_RNS_PB[PB_CmdPause].LampON;
END_ACTION
```

#### RNS_StepManager.st
```iecst
ACTION RNS_StepManager:
	//PROD
	VAR_RNS_SeqProdStopAlarm := VAR_RNS_AVB_ValveFault OR
								VAR_RNS_WaterFlowTooLow OR VAR_RNS_WaterFlowMissing ;

	IF VAR_RNS_SeqProdStopAlarm THEN
		VAR_RNS_SeqProdStopRequest	:= VAR_RNS_ModeProduction;
	END_IF

	IF VAR_RNS_StepProdStopped OR VAR_RNS_StepProdLampOnDischarge THEN
		VAR_RNS_SeqProdStopRequest	:= FALSE;
	END_IF

	IF VAR_RNS_MemPBStop OR NOT VAR_RNS_FMDProduction THEN //SEQUENCE ABORT IS MANAGED BY STOP PB or finish tank process
		VAR_RNS_SeqProdAbortRequest	:= VAR_RNS_ModeProduction;
	END_IF
	IF VAR_RNS_StepProdAborted THEN
		VAR_RNS_SeqProdAbortRequest	:= FALSE;
	END_IF

	//CIP
//	VAR_RNS_SeqCipStopAlarm := NOT OPS.DataOut.EmergencyOk OR NOT OPS.DataOut.DoorsOk OR VAR_RNS_AVB_ValveFault;

	IF  VAR_RNS_SeqCipStopAlarm THEN
		VAR_RNS_SeqCipStopRequest	:= VAR_RNS_ModeCip;
	END_IF
	IF VAR_RNS_StepCipStopped THEN
		VAR_RNS_SeqCipStopRequest	:= FALSE;
	END_IF

	IF  VAR_RNS_MemPBStop OR NOT VAR_RNS_FMDCip THEN //SEQUENCE ABORT IS MANAGED BY STOP PB
		VAR_RNS_SeqCipAbortRequest	:= VAR_RNS_ModeCip;
	END_IF
	IF VAR_RNS_StepCipAborted THEN
		VAR_RNS_SeqCipAbortRequest	:= FALSE;
	END_IF

	//DRAIN
	VAR_RNS_SeqDrainStopAlarm := NOT OPS.DataOut.EmergencyOk OR NOT OPS.DataOut.DoorsOk OR VAR_RNS_AVB_ValveFault;

	IF VAR_RNS_SeqDrainStopAlarm THEN
		VAR_RNS_SeqDrainStopRequest	:= VAR_RNS_ModeDrain;
	END_IF
	IF VAR_RNS_StepDrainStopped THEN
		VAR_RNS_SeqDrainStopRequest	:= FALSE;
	END_IF

	IF VAR_RNS_MemPBStop OR NOT VAR_RNS_FMDDrain THEN //SEQUENCE ABORT IS MANAGED BY STOP PB
		VAR_RNS_SeqDrainAbortRequest := VAR_RNS_ModeDrain;
	END_IF
	IF VAR_RNS_StepDrainAborted THEN
		VAR_RNS_SeqDrainAbortRequest := FALSE;
	END_IF

	//CONTROL
	VAR_RNS_SeqControlStopAlarm := 	NOT OPS.DataOut.EmergencyOk OR NOT OPS.DataOut.DoorsOk OR VAR_RNS_AVB_ValveFault OR
									VAR_RNS_WaterFlowTooLow OR VAR_RNS_AirFlowTooLow OR VAR_RNS_WaterFlowMissing;

	IF VAR_RNS_SeqControlStopAlarm THEN
		VAR_RNS_SeqControlStopRequest	:= VAR_RNS_ModeControl;
	END_IF
	IF VAR_RNS_StepControlStopped THEN
		VAR_RNS_SeqControlStopRequest	:= FALSE;
	END_IF

	IF VAR_RNS_MemPBStop THEN //SEQUENCE ABORT IS MANAGED BY STOP PB
		VAR_RNS_SeqControlAbortRequest := VAR_RNS_ModeControl;
	END_IF
	IF VAR_RNS_StepControlAborted THEN
		VAR_RNS_SeqControlAbortRequest := FALSE;
	END_IF

END_ACTION
```
